// TwinCAT 3 PLC project Walking_Welding_Robot_Control_System
// ProgramVersion: 3.1.4020.4
// libraries:
//   Tc2_MC2, * (Beckhoff Automation GmbH)
//   Tc2_Standard, * (Beckhoff Automation GmbH)
//   Tc2_System, * (Beckhoff Automation GmbH)
//   Tc3_Module, * (Beckhoff Automation GmbH)
//   VisuDialogs, * (System)
// project tree:
//   DUTs/Axis/ Axis.TcPOU
//   DUTs/Filter_Current/ FB_Filter_Current_Hexapod_Robot.TcPOU, ST_Filter_Current_Hexapod_Robot_InitData.TcDUT, ST_Filter_Current_Hexapod_Robot_Input.TcDUT, ST_Filter_Current_Hexapod_Robot_Output.TcDUT
//   DUTs/Hexapod_Leg/ Hexapod_Leg.TcPOU (not stored)
//   DUTs/Mapping/ Leg_Control_Mapping_Model.TcPOU (not stored), Leg_Model_Mapping_Control.TcPOU (not stored), Variable_Control_Mapping_Model.TcPOU (not stored), Variable_Model_Mapping_Control.TcPOU (not stored)
//   DUTs/Robot_Simulink/ E_TcMatSimDataAreaType.TcDUT (not stored), FB_RobotWalking_OnEvenTerrain.TcPOU (not stored), FB_TcMatSimObject.TcPOU (not stored), ST_RobotWalking_OnEvenTerrain_InitData.TcDUT (not stored), ST_RobotWalking_OnEvenTerrain_Input.TcDUT (not stored), ST_RobotWalking_OnEvenTerrain_Output.TcDUT (not stored), ST_TcMatSimObjectDataAreaInfo.TcDUT (not stored)
//   DUTs/Touch_Signal_Detection/ FB_Tough_Signal_Detection_Simple.TcPOU, ST_Tough_Signal_Detection_Simple_InitData.TcDUT, ST_Tough_Signal_Detection_Simple_Input.TcDUT, ST_Tough_Signal_Detection_Simple_Output.TcDUT
//   DUTs/Welding_Arm_Simulink/ FB_WeldingArm6AxisMotion_Control.TcPOU, ST_WeldingArm6AxisMotion_Control_InitData.TcDUT, ST_WeldingArm6AxisMotion_Control_Input.TcDUT, ST_WeldingArm6AxisMotion_Control_Output.TcDUT
//   / GlobalTextList.TcGTLO, PlcTask.TcTTO, Sensor_Test.TcTTO, Simulink_Test.TcTTO, 视图管理器.TcVMO (not stored)
//   POUs/ Walking_Robot_Control.TcPOU, SignalData_Interface.TcPOU, Walking_Robot_Movement.TcPOU, Walking_Welding_Robot_Control.TcPOU, Welding_Arm_Control.TcPOU, Welding_Arm_Movement.TcPOU
//   VISUs/ ImagePool.TcIPO (not stored), Visu_Welding_Arm_Power.TcVIS, Visu_Welding_Arm_SimulinkMove.TcVIS, Visu_Walking_Robot_Home.TcVIS, Visu_Walking_Robot_Power.TcVIS, Visu_Walking_Robot_Reset.TcVIS, Visu_Walking_Robot_SimulinkMove.TcVIS, Visu_Walking_Robot_Stand.TcVIS, Visu_Walking_Welding_Robot_Control.TcVIS, Visu_Welcome.TcVIS, Visu_Welding_Arm_OldVersion.TcVIS
// real-time tasks:
//   TASK PlcTask: cycle T#4ms, priority 12, ADS port 350
//   TASK Simulink_Test: cycle T#4ms, priority 6, ADS port 351
//   TASK Sensor_Test: cycle T#1ms, priority 14, ADS port 352
//   TASK Walking_Welding_Robot_Task: cycle T#4ms, priority 10, ADS port 353
// motion (NC):
//   TASK NC-Task 1 SAF: cycle T#4ms, priority 4, ADS port 501
//   TASK NC-Task 1 SVB: cycle T#4ms, priority 8, ADS port 511
//   AXIS Axis 1 (id 1)
//     Velo: SlowManual=10, FastManual=20
//     OtherSettings: AllowMotionCmdToSlave=true, AllowMotionCmdToExtSetGenAxis=true
//     encoder EncType=19
//       EncPara: ScaleFactorNumerator=0.000152590218967, MaxCount=#xffffffff
//     drive DrvType=16
//       DrvPara: MaxCount=#xffffffff
//         TimeComp: TaskDelayCycles=1
//     controller CtrType=1
//       CtrPara: PriorControlFactor=1
//         Observer: BandWidth=20
//   AXIS Axis 2 (id 2)
//     Velo: SlowManual=10, FastManual=20
//     OtherSettings: AllowMotionCmdToSlave=true, AllowMotionCmdToExtSetGenAxis=true
//     encoder EncType=19
//       EncPara: ScaleFactorNumerator=0.000152590218967, MaxCount=#xffffffff
//     drive DrvType=16
//       DrvPara: MaxCount=#xffffffff
//         TimeComp: TaskDelayCycles=1
//     controller CtrType=1
//       CtrPara: PriorControlFactor=1
//         Observer: BandWidth=20
//   AXIS Axis 3 (id 3)
//     Velo: SlowManual=10, FastManual=20
//     OtherSettings: AllowMotionCmdToSlave=true, AllowMotionCmdToExtSetGenAxis=true
//     encoder EncType=19
//       EncPara: ScaleFactorNumerator=0.000152590218967, MaxCount=#xffffffff
//     drive DrvType=16
//       DrvPara: MaxCount=#xffffffff
//         TimeComp: TaskDelayCycles=1
//     controller CtrType=1
//       CtrPara: PriorControlFactor=1
//         Observer: BandWidth=20
//   AXIS Axis 4 (id 4)
//     Velo: SlowManual=10, FastManual=20
//     OtherSettings: AllowMotionCmdToSlave=true, AllowMotionCmdToExtSetGenAxis=true
//     encoder EncType=19
//       EncPara: ScaleFactorNumerator=0.000152590218967, MaxCount=#xffffffff
//     drive DrvType=16
//       DrvPara: MaxCount=#xffffffff
//         TimeComp: TaskDelayCycles=1
//     controller CtrType=1
//       CtrPara: PriorControlFactor=1
//         Observer: BandWidth=20
//   AXIS Axis 5 (id 5)
//     Velo: SlowManual=10, FastManual=20
//     OtherSettings: AllowMotionCmdToSlave=true, AllowMotionCmdToExtSetGenAxis=true
//     encoder EncType=19
//       EncPara: ScaleFactorNumerator=0.000152590218967, MaxCount=#xffffffff
//     drive DrvType=16
//       DrvPara: MaxCount=#xffffffff
//         TimeComp: TaskDelayCycles=1
//     controller CtrType=1
//       CtrPara: PriorControlFactor=1
//         Observer: BandWidth=20
//   AXIS Axis 6 (id 6)
//     Velo: SlowManual=10, FastManual=20
//     OtherSettings: AllowMotionCmdToSlave=true, AllowMotionCmdToExtSetGenAxis=true
//     encoder EncType=19
//       EncPara: ScaleFactorNumerator=0.000152590218967, MaxCount=#xffffffff
//     drive DrvType=16
//       DrvPara: MaxCount=#xffffffff
//         TimeComp: TaskDelayCycles=1
//     controller CtrType=1
//       CtrPara: PriorControlFactor=1
//         Observer: BandWidth=20
//   AXIS Axis 7 (id 7)
//     Velo: SlowManual=10, FastManual=20
//     OtherSettings: AllowMotionCmdToSlave=true, AllowMotionCmdToExtSetGenAxis=true
//     encoder EncType=19
//       EncPara: ScaleFactorNumerator=0.000152590218967, MaxCount=#xffffffff
//     drive DrvType=16
//       DrvPara: MaxCount=#xffffffff
//         TimeComp: TaskDelayCycles=1
//     controller CtrType=1
//       CtrPara: PriorControlFactor=1
//         Observer: BandWidth=20
//   AXIS Axis 8 (id 8)
//     Velo: SlowManual=10, FastManual=20
//     OtherSettings: AllowMotionCmdToSlave=true, AllowMotionCmdToExtSetGenAxis=true
//     encoder EncType=19
//       EncPara: ScaleFactorNumerator=0.000152590218967, MaxCount=#xffffffff
//     drive DrvType=16
//       DrvPara: MaxCount=#xffffffff
//         TimeComp: TaskDelayCycles=1
//     controller CtrType=1
//       CtrPara: PriorControlFactor=1
//         Observer: BandWidth=20
//   AXIS Axis 9 (id 9)
//     Velo: SlowManual=10, FastManual=20
//     OtherSettings: AllowMotionCmdToSlave=true, AllowMotionCmdToExtSetGenAxis=true
//     encoder EncType=19
//       EncPara: ScaleFactorNumerator=0.000152590218967, MaxCount=#xffffffff
//     drive DrvType=16
//       DrvPara: MaxCount=#xffffffff
//         TimeComp: TaskDelayCycles=1
//     controller CtrType=1
//       CtrPara: PriorControlFactor=1
//         Observer: BandWidth=20
//   AXIS Axis 10 (id 10)
//     Velo: SlowManual=10, FastManual=20
//     OtherSettings: AllowMotionCmdToSlave=true, AllowMotionCmdToExtSetGenAxis=true
//     encoder EncType=19
//       EncPara: ScaleFactorNumerator=0.000152590218967, MaxCount=#xffffffff
//     drive DrvType=16
//       DrvPara: MaxCount=#xffffffff
//         TimeComp: TaskDelayCycles=1
//     controller CtrType=1
//       CtrPara: PriorControlFactor=1
//         Observer: BandWidth=20
//   AXIS Axis 11 (id 11)
//     Velo: SlowManual=10, FastManual=20
//     OtherSettings: AllowMotionCmdToSlave=true, AllowMotionCmdToExtSetGenAxis=true
//     encoder EncType=19
//       EncPara: ScaleFactorNumerator=0.000152590218967, MaxCount=#xffffffff
//     drive DrvType=16
//       DrvPara: MaxCount=#xffffffff
//         TimeComp: TaskDelayCycles=1
//     controller CtrType=1
//       CtrPara: PriorControlFactor=1
//         Observer: BandWidth=20
//   AXIS Axis 12 (id 12)
//     Velo: SlowManual=10, FastManual=20
//     OtherSettings: AllowMotionCmdToSlave=true, AllowMotionCmdToExtSetGenAxis=true
//     encoder EncType=19
//       EncPara: ScaleFactorNumerator=0.000152590218967, MaxCount=#xffffffff
//     drive DrvType=16
//       DrvPara: MaxCount=#xffffffff
//         TimeComp: TaskDelayCycles=1
//     controller CtrType=1
//       CtrPara: PriorControlFactor=1
//         Observer: BandWidth=20
//   AXIS Axis 13 (id 13)
//     Velo: SlowManual=10, FastManual=20
//     OtherSettings: AllowMotionCmdToSlave=true, AllowMotionCmdToExtSetGenAxis=true
//     encoder EncType=19
//       EncPara: ScaleFactorNumerator=0.000152590218967, MaxCount=#xffffffff
//     drive DrvType=16
//       DrvPara: MaxCount=#xffffffff
//         TimeComp: TaskDelayCycles=1
//     controller CtrType=1
//       CtrPara: PriorControlFactor=1
//         Observer: BandWidth=20
//   AXIS Axis 14 (id 14)
//     Velo: SlowManual=10, FastManual=20
//     OtherSettings: AllowMotionCmdToSlave=true, AllowMotionCmdToExtSetGenAxis=true
//     encoder EncType=19
//       EncPara: ScaleFactorNumerator=0.000152590218967, MaxCount=#xffffffff
//     drive DrvType=16
//       DrvPara: MaxCount=#xffffffff
//         TimeComp: TaskDelayCycles=1
//     controller CtrType=1
//       CtrPara: PriorControlFactor=1
//         Observer: BandWidth=20
//   AXIS Axis 15 (id 15)
//     Velo: SlowManual=10, FastManual=20
//     OtherSettings: AllowMotionCmdToSlave=true, AllowMotionCmdToExtSetGenAxis=true
//     encoder EncType=19
//       EncPara: ScaleFactorNumerator=0.000152590218967, MaxCount=#xffffffff
//     drive DrvType=16
//       DrvPara: MaxCount=#xffffffff
//         TimeComp: TaskDelayCycles=1
//     controller CtrType=1
//       CtrPara: PriorControlFactor=1
//         Observer: BandWidth=20
//   AXIS Axis 16 (id 16)
//     Velo: SlowManual=10, FastManual=20
//     OtherSettings: AllowMotionCmdToSlave=true, AllowMotionCmdToExtSetGenAxis=true
//     encoder EncType=19
//       EncPara: ScaleFactorNumerator=0.000152590218967, MaxCount=#xffffffff
//     drive DrvType=16
//       DrvPara: MaxCount=#xffffffff
//         TimeComp: TaskDelayCycles=1
//     controller CtrType=1
//       CtrPara: PriorControlFactor=1
//         Observer: BandWidth=20
//   AXIS Axis 17 (id 17)
//     Velo: SlowManual=10, FastManual=20
//     OtherSettings: AllowMotionCmdToSlave=true, AllowMotionCmdToExtSetGenAxis=true
//     encoder EncType=19
//       EncPara: ScaleFactorNumerator=0.000152590218967, MaxCount=#xffffffff
//     drive DrvType=16
//       DrvPara: MaxCount=#xffffffff
//         TimeComp: TaskDelayCycles=1
//     controller CtrType=1
//       CtrPara: PriorControlFactor=1
//         Observer: BandWidth=20
//   AXIS Axis 18 (id 18)
//     Velo: SlowManual=10, FastManual=20
//     OtherSettings: AllowMotionCmdToSlave=true, AllowMotionCmdToExtSetGenAxis=true
//     encoder EncType=19
//       EncPara: ScaleFactorNumerator=0.000152590218967, MaxCount=#xffffffff
//     drive DrvType=16
//       DrvPara: MaxCount=#xffffffff
//         TimeComp: TaskDelayCycles=1
//     controller CtrType=1
//       CtrPara: PriorControlFactor=1
//         Observer: BandWidth=20
//   AXIS Axis 19 (id 19)
//     Velo: SlowManual=10, FastManual=20
//     OtherSettings: AllowMotionCmdToSlave=true
//     encoder EncType=19
//       EncPara: ScaleFactorNumerator=1.6954468774e-005, MaxCount=#xffffffff
//     drive DrvType=16
//       DrvPara: MaxCount=#xffffffff
//         TimeComp: TaskDelayCycles=1
//     controller CtrType=1
//       CtrPara: PriorControlFactor=1
//         Observer: BandWidth=20
//   AXIS Axis 20 (id 20)
//     Velo: SlowManual=10, FastManual=20
//     OtherSettings: AllowMotionCmdToSlave=true
//     encoder EncType=19
//       EncPara: ScaleFactorNumerator=0.006206896551724, MaxCount=#xffffffff
//     drive DrvType=16
//       DrvPara: MaxCount=#xffffffff
//         TimeComp: TaskDelayCycles=1
//     controller CtrType=1
//       CtrPara: PriorControlFactor=1
//         Observer: BandWidth=20
//   AXIS Axis 21 (id 21)
//     Velo: SlowManual=10, FastManual=20
//     OtherSettings: AllowMotionCmdToSlave=true
//     encoder EncType=19
//       EncPara: ScaleFactorNumerator=2.441443503e-006, MaxCount=#xffffffff
//     drive DrvType=16
//       DrvPara: MaxCount=#xffffffff
//         TimeComp: TaskDelayCycles=1
//     controller CtrType=1
//       CtrPara: PriorControlFactor=1
//         Observer: BandWidth=20
//   AXIS Axis 22 (id 22)
//     Velo: SlowManual=10, FastManual=20
//     OtherSettings: AllowMotionCmdToSlave=true
//     encoder EncType=19
//       EncPara: ScaleFactorNumerator=0.000365910901229, MaxCount=#xffffffff
//     drive DrvType=16
//       DrvPara: MaxCount=#xffffffff
//         TimeComp: TaskDelayCycles=1
//     controller CtrType=1
//       CtrPara: PriorControlFactor=1
//         Observer: BandWidth=20
//   AXIS Axis 23 (id 23)
//     Velo: SlowManual=10, FastManual=20
//     OtherSettings: AllowMotionCmdToSlave=true
//     encoder EncType=19
//       EncPara: ScaleFactorNumerator=0.000365910901229, MaxCount=#xffffffff
//     drive DrvType=16
//       DrvPara: MaxCount=#xffffffff
//         TimeComp: TaskDelayCycles=1
//     controller CtrType=1
//       CtrPara: PriorControlFactor=1
//         Observer: BandWidth=20
//   AXIS Axis 24 (id 24)
//     Velo: SlowManual=10, FastManual=20
//     OtherSettings: AllowMotionCmdToSlave=true
//     encoder EncType=19
//       EncPara: ScaleFactorNumerator=0.000365910901229, MaxCount=#xffffffff
//     drive DrvType=16
//       DrvPara: MaxCount=#xffffffff
//         TimeComp: TaskDelayCycles=1
//     controller CtrType=1
//       CtrPara: PriorControlFactor=1
//         Observer: BandWidth=20
// I/O:
//   DEVICE Device 3 (EtherCAT), AmsNetId 5.41.150.106.4.1
//     Drive 1 (Elmo Drive) [Gold EtherCAT GCON Drive Rev:0x000103F6]
//     Drive 2 (Elmo Drive) [Gold EtherCAT GCON Drive Rev:0x000103F6]
//     Drive 3 (Elmo Drive) [Gold EtherCAT GCON Drive Rev:0x000103F6]
//     Drive 4 (Elmo Drive) [Gold EtherCAT GCON Drive Rev:0x000103F6]
//     Drive 5 (Elmo Drive) [Gold EtherCAT GCON Drive Rev:0x000103F6]
//     Drive 6 (Elmo Drive) [Gold EtherCAT GCON Drive Rev:0x000103F6]
//     Drive 7 (Elmo Drive) [Gold EtherCAT GCON Drive Rev:0x000103F6]
//     Drive 8 (Elmo Drive) [Gold EtherCAT GCON Drive Rev:0x000103F6]
//     Drive 9 (Elmo Drive) [Gold EtherCAT GCON Drive Rev:0x000103F6]
//     Drive 10 (Elmo Drive) [Gold EtherCAT GCON Drive Rev:0x000103F6]
//     Drive 11 (Elmo Drive) [Gold EtherCAT GCON Drive Rev:0x000103F6]
//     Drive 12 (Elmo Drive) [Gold EtherCAT GCON Drive Rev:0x000103F6]
//     Drive 13 (Elmo Drive) [Gold EtherCAT GCON Drive Rev:0x000103F6]
//     Drive 14 (Elmo Drive) [Gold EtherCAT GCON Drive Rev:0x000103F6]
//     Drive 15 (Elmo Drive) [Gold EtherCAT GCON Drive Rev:0x000103F6]
//     Drive 16 (Elmo Drive) [Gold EtherCAT GCON Drive Rev:0x000103F6]
//     Drive 17 (Elmo Drive) [Gold EtherCAT GCON Drive Rev:0x000103F6]
//     Drive 18 (Elmo Drive) [Gold EtherCAT GCON Drive Rev:0x000103F6]
//     Drive 37 (Elmo Drive) [Gold EtherCAT GCON Drive Rev:0x000103F6]
//     Drive 38 (Elmo Drive) [Gold EtherCAT GCON Drive Rev:0x000103F6]
//     Drive 39 (Elmo Drive) [Gold EtherCAT GCON Drive Rev:0x000103F6]
//     Drive 40 (Elmo Drive) [Gold EtherCAT GCON Drive Rev:0x000103F6]
//     Drive 41 (Elmo Drive) [Gold EtherCAT GCON Drive Rev:0x000103F6]
//     Drive 42 (Elmo Drive) [Gold EtherCAT GCON Drive Rev:0x000103F6]
// variable links:
//   NC-Task 1 SAF/Axes/Axis 1 <-> Device 3 (EtherCAT)/Drive 1 (Elmo Drive)
//     Drive/Inputs/In/nDcOutputTime <-> InfoData/DcOutputShift
//     Drive/Inputs/In/nState1 <-> Inputs/Status word
//     Drive/Inputs/In/nState2 <-> Inputs/Status word @bit 8
//     Drive/Inputs/In/nState4 @bit 1 <-> WcState/InputToggle
//     Drive/Inputs/In/nState4 <-> WcState/WcState
//     Drive/Outputs/Out/nCtrl1 <-> Outputs/Control word
//     Drive/Outputs/Out/nCtrl2 <-> Outputs/Control word @bit 8
//     Drive/Outputs/Out/nDataOut1 <-> Outputs/Target Position
//     Enc/Inputs/In/nDataIn1 <-> Inputs/Position actual value
//     Enc/Inputs/In/nDcInputTime <-> InfoData/DcInputShift
//     Enc/Inputs/In/nState4 @bit 1 <-> WcState/InputToggle
//     Enc/Inputs/In/nState4 <-> WcState/WcState
//   NC-Task 1 SAF/Axes/Axis 10 <-> Device 3 (EtherCAT)/Drive 10 (Elmo Drive)
//     Drive/Inputs/In/nDcOutputTime <-> InfoData/DcOutputShift
//     Drive/Inputs/In/nState1 <-> Inputs/Status word
//     Drive/Inputs/In/nState2 <-> Inputs/Status word @bit 8
//     Drive/Inputs/In/nState4 @bit 1 <-> WcState/InputToggle
//     Drive/Inputs/In/nState4 <-> WcState/WcState
//     Drive/Outputs/Out/nCtrl1 <-> Outputs/Control word
//     Drive/Outputs/Out/nCtrl2 <-> Outputs/Control word @bit 8
//     Drive/Outputs/Out/nDataOut1 <-> Outputs/Target Position
//     Enc/Inputs/In/nDataIn1 <-> Inputs/Position actual value
//     Enc/Inputs/In/nDcInputTime <-> InfoData/DcInputShift
//     Enc/Inputs/In/nState4 @bit 1 <-> WcState/InputToggle
//     Enc/Inputs/In/nState4 <-> WcState/WcState
//   NC-Task 1 SAF/Axes/Axis 11 <-> Device 3 (EtherCAT)/Drive 11 (Elmo Drive)
//     Drive/Inputs/In/nDcOutputTime <-> InfoData/DcOutputShift
//     Drive/Inputs/In/nState1 <-> Inputs/Status word
//     Drive/Inputs/In/nState2 <-> Inputs/Status word @bit 8
//     Drive/Inputs/In/nState4 @bit 1 <-> WcState/InputToggle
//     Drive/Inputs/In/nState4 <-> WcState/WcState
//     Drive/Outputs/Out/nCtrl1 <-> Outputs/Control word
//     Drive/Outputs/Out/nCtrl2 <-> Outputs/Control word @bit 8
//     Drive/Outputs/Out/nDataOut1 <-> Outputs/Target Position
//     Enc/Inputs/In/nDataIn1 <-> Inputs/Position actual value
//     Enc/Inputs/In/nDcInputTime <-> InfoData/DcInputShift
//     Enc/Inputs/In/nState4 @bit 1 <-> WcState/InputToggle
//     Enc/Inputs/In/nState4 <-> WcState/WcState
//   NC-Task 1 SAF/Axes/Axis 12 <-> Device 3 (EtherCAT)/Drive 12 (Elmo Drive)
//     Drive/Inputs/In/nDcOutputTime <-> InfoData/DcOutputShift
//     Drive/Inputs/In/nState1 <-> Inputs/Status word
//     Drive/Inputs/In/nState2 <-> Inputs/Status word @bit 8
//     Drive/Inputs/In/nState4 @bit 1 <-> WcState/InputToggle
//     Drive/Inputs/In/nState4 <-> WcState/WcState
//     Drive/Outputs/Out/nCtrl1 <-> Outputs/Control word
//     Drive/Outputs/Out/nCtrl2 <-> Outputs/Control word @bit 8
//     Drive/Outputs/Out/nDataOut1 <-> Outputs/Target Position
//     Enc/Inputs/In/nDataIn1 <-> Inputs/Position actual value
//     Enc/Inputs/In/nDcInputTime <-> InfoData/DcInputShift
//     Enc/Inputs/In/nState4 @bit 1 <-> WcState/InputToggle
//     Enc/Inputs/In/nState4 <-> WcState/WcState
//   NC-Task 1 SAF/Axes/Axis 13 <-> Device 3 (EtherCAT)/Drive 13 (Elmo Drive)
//     Drive/Inputs/In/nDcOutputTime <-> InfoData/DcOutputShift
//     Drive/Inputs/In/nState1 <-> Inputs/Status word
//     Drive/Inputs/In/nState2 <-> Inputs/Status word @bit 8
//     Drive/Inputs/In/nState4 @bit 1 <-> WcState/InputToggle
//     Drive/Inputs/In/nState4 <-> WcState/WcState
//     Drive/Outputs/Out/nCtrl1 <-> Outputs/Control word
//     Drive/Outputs/Out/nCtrl2 <-> Outputs/Control word @bit 8
//     Drive/Outputs/Out/nDataOut1 <-> Outputs/Target Position
//     Enc/Inputs/In/nDataIn1 <-> Inputs/Position actual value
//     Enc/Inputs/In/nDcInputTime <-> InfoData/DcInputShift
//     Enc/Inputs/In/nState4 @bit 1 <-> WcState/InputToggle
//     Enc/Inputs/In/nState4 <-> WcState/WcState
//   NC-Task 1 SAF/Axes/Axis 14 <-> Device 3 (EtherCAT)/Drive 14 (Elmo Drive)
//     Drive/Inputs/In/nDcOutputTime <-> InfoData/DcOutputShift
//     Drive/Inputs/In/nState1 <-> Inputs/Status word
//     Drive/Inputs/In/nState2 <-> Inputs/Status word @bit 8
//     Drive/Inputs/In/nState4 @bit 1 <-> WcState/InputToggle
//     Drive/Inputs/In/nState4 <-> WcState/WcState
//     Drive/Outputs/Out/nCtrl1 <-> Outputs/Control word
//     Drive/Outputs/Out/nCtrl2 <-> Outputs/Control word @bit 8
//     Drive/Outputs/Out/nDataOut1 <-> Outputs/Target Position
//     Enc/Inputs/In/nDataIn1 <-> Inputs/Position actual value
//     Enc/Inputs/In/nDcInputTime <-> InfoData/DcInputShift
//     Enc/Inputs/In/nState4 @bit 1 <-> WcState/InputToggle
//     Enc/Inputs/In/nState4 <-> WcState/WcState
//   NC-Task 1 SAF/Axes/Axis 15 <-> Device 3 (EtherCAT)/Drive 15 (Elmo Drive)
//     Drive/Inputs/In/nDcOutputTime <-> InfoData/DcOutputShift
//     Drive/Inputs/In/nState1 <-> Inputs/Status word
//     Drive/Inputs/In/nState2 <-> Inputs/Status word @bit 8
//     Drive/Inputs/In/nState4 @bit 1 <-> WcState/InputToggle
//     Drive/Inputs/In/nState4 <-> WcState/WcState
//     Drive/Outputs/Out/nCtrl1 <-> Outputs/Control word
//     Drive/Outputs/Out/nCtrl2 <-> Outputs/Control word @bit 8
//     Drive/Outputs/Out/nDataOut1 <-> Outputs/Target Position
//     Enc/Inputs/In/nDataIn1 <-> Inputs/Position actual value
//     Enc/Inputs/In/nDcInputTime <-> InfoData/DcInputShift
//     Enc/Inputs/In/nState4 @bit 1 <-> WcState/InputToggle
//     Enc/Inputs/In/nState4 <-> WcState/WcState
//   NC-Task 1 SAF/Axes/Axis 16 <-> Device 3 (EtherCAT)/Drive 16 (Elmo Drive)
//     Drive/Inputs/In/nDcOutputTime <-> InfoData/DcOutputShift
//     Drive/Inputs/In/nState1 <-> Inputs/Status word
//     Drive/Inputs/In/nState2 <-> Inputs/Status word @bit 8
//     Drive/Inputs/In/nState4 @bit 1 <-> WcState/InputToggle
//     Drive/Inputs/In/nState4 <-> WcState/WcState
//     Drive/Outputs/Out/nCtrl1 <-> Outputs/Control word
//     Drive/Outputs/Out/nCtrl2 <-> Outputs/Control word @bit 8
//     Drive/Outputs/Out/nDataOut1 <-> Outputs/Target Position
//     Enc/Inputs/In/nDataIn1 <-> Inputs/Position actual value
//     Enc/Inputs/In/nDcInputTime <-> InfoData/DcInputShift
//     Enc/Inputs/In/nState4 @bit 1 <-> WcState/InputToggle
//     Enc/Inputs/In/nState4 <-> WcState/WcState
//   NC-Task 1 SAF/Axes/Axis 17 <-> Device 3 (EtherCAT)/Drive 17 (Elmo Drive)
//     Drive/Inputs/In/nDcOutputTime <-> InfoData/DcOutputShift
//     Drive/Inputs/In/nState1 <-> Inputs/Status word
//     Drive/Inputs/In/nState2 <-> Inputs/Status word @bit 8
//     Drive/Inputs/In/nState4 @bit 1 <-> WcState/InputToggle
//     Drive/Inputs/In/nState4 <-> WcState/WcState
//     Drive/Outputs/Out/nCtrl1 <-> Outputs/Control word
//     Drive/Outputs/Out/nCtrl2 <-> Outputs/Control word @bit 8
//     Drive/Outputs/Out/nDataOut1 <-> Outputs/Target Position
//     Enc/Inputs/In/nDataIn1 <-> Inputs/Position actual value
//     Enc/Inputs/In/nDcInputTime <-> InfoData/DcInputShift
//     Enc/Inputs/In/nState4 @bit 1 <-> WcState/InputToggle
//     Enc/Inputs/In/nState4 <-> WcState/WcState
//   NC-Task 1 SAF/Axes/Axis 18 <-> Device 3 (EtherCAT)/Drive 18 (Elmo Drive)
//     Drive/Inputs/In/nDcOutputTime <-> InfoData/DcOutputShift
//     Drive/Inputs/In/nState1 <-> Inputs/Status word
//     Drive/Inputs/In/nState2 <-> Inputs/Status word @bit 8
//     Drive/Inputs/In/nState4 @bit 1 <-> WcState/InputToggle
//     Drive/Inputs/In/nState4 <-> WcState/WcState
//     Drive/Outputs/Out/nCtrl1 <-> Outputs/Control word
//     Drive/Outputs/Out/nCtrl2 <-> Outputs/Control word @bit 8
//     Drive/Outputs/Out/nDataOut1 <-> Outputs/Target Position
//     Enc/Inputs/In/nDataIn1 <-> Inputs/Position actual value
//     Enc/Inputs/In/nDcInputTime <-> InfoData/DcInputShift
//     Enc/Inputs/In/nState4 @bit 1 <-> WcState/InputToggle
//     Enc/Inputs/In/nState4 <-> WcState/WcState
//   NC-Task 1 SAF/Axes/Axis 19 <-> Device 3 (EtherCAT)/Drive 37 (Elmo Drive)
//     Drive/Inputs/In/nDcOutputTime <-> InfoData/DcOutputShift
//     Drive/Inputs/In/nState1 <-> Inputs/Status word
//     Drive/Inputs/In/nState2 <-> Inputs/Status word @bit 8
//     Drive/Inputs/In/nState4 @bit 1 <-> WcState/InputToggle
//     Drive/Inputs/In/nState4 <-> WcState/WcState
//     Drive/Outputs/Out/nCtrl1 <-> Outputs/Control word
//     Drive/Outputs/Out/nCtrl2 <-> Outputs/Control word @bit 8
//     Drive/Outputs/Out/nDataOut1 <-> Outputs/Target Position
//     Enc/Inputs/In/nDataIn1 <-> Inputs/Position actual value
//     Enc/Inputs/In/nDcInputTime <-> InfoData/DcInputShift
//     Enc/Inputs/In/nState4 @bit 1 <-> WcState/InputToggle
//     Enc/Inputs/In/nState4 <-> WcState/WcState
//   NC-Task 1 SAF/Axes/Axis 2 <-> Device 3 (EtherCAT)/Drive 2 (Elmo Drive)
//     Drive/Inputs/In/nDcOutputTime <-> InfoData/DcOutputShift
//     Drive/Inputs/In/nState1 <-> Inputs/Status word
//     Drive/Inputs/In/nState2 <-> Inputs/Status word @bit 8
//     Drive/Inputs/In/nState4 @bit 1 <-> WcState/InputToggle
//     Drive/Inputs/In/nState4 <-> WcState/WcState
//     Drive/Outputs/Out/nCtrl1 <-> Outputs/Control word
//     Drive/Outputs/Out/nCtrl2 <-> Outputs/Control word @bit 8
//     Drive/Outputs/Out/nDataOut1 <-> Outputs/Target Position
//     Enc/Inputs/In/nDataIn1 <-> Inputs/Position actual value
//     Enc/Inputs/In/nDcInputTime <-> InfoData/DcInputShift
//     Enc/Inputs/In/nState4 @bit 1 <-> WcState/InputToggle
//     Enc/Inputs/In/nState4 <-> WcState/WcState
//   NC-Task 1 SAF/Axes/Axis 20 <-> Device 3 (EtherCAT)/Drive 38 (Elmo Drive)
//     Drive/Inputs/In/nDcOutputTime <-> InfoData/DcOutputShift
//     Drive/Inputs/In/nState1 <-> Inputs/Status word
//     Drive/Inputs/In/nState2 <-> Inputs/Status word @bit 8
//     Drive/Inputs/In/nState4 @bit 1 <-> WcState/InputToggle
//     Drive/Inputs/In/nState4 <-> WcState/WcState
//     Drive/Outputs/Out/nCtrl1 <-> Outputs/Control word
//     Drive/Outputs/Out/nCtrl2 <-> Outputs/Control word @bit 8
//     Drive/Outputs/Out/nDataOut1 <-> Outputs/Target Position
//     Enc/Inputs/In/nDataIn1 <-> Inputs/Position actual value
//     Enc/Inputs/In/nDcInputTime <-> InfoData/DcInputShift
//     Enc/Inputs/In/nState4 @bit 1 <-> WcState/InputToggle
//     Enc/Inputs/In/nState4 <-> WcState/WcState
//   NC-Task 1 SAF/Axes/Axis 21 <-> Device 3 (EtherCAT)/Drive 39 (Elmo Drive)
//     Drive/Inputs/In/nDcOutputTime <-> InfoData/DcOutputShift
//     Drive/Inputs/In/nState1 <-> Inputs/Status word
//     Drive/Inputs/In/nState2 <-> Inputs/Status word @bit 8
//     Drive/Inputs/In/nState4 @bit 1 <-> WcState/InputToggle
//     Drive/Inputs/In/nState4 <-> WcState/WcState
//     Drive/Outputs/Out/nCtrl1 <-> Outputs/Control word
//     Drive/Outputs/Out/nCtrl2 <-> Outputs/Control word @bit 8
//     Drive/Outputs/Out/nDataOut1 <-> Outputs/Target Position
//     Enc/Inputs/In/nDataIn1 <-> Inputs/Position actual value
//     Enc/Inputs/In/nDcInputTime <-> InfoData/DcInputShift
//     Enc/Inputs/In/nState4 @bit 1 <-> WcState/InputToggle
//     Enc/Inputs/In/nState4 <-> WcState/WcState
//   NC-Task 1 SAF/Axes/Axis 22 <-> Device 3 (EtherCAT)/Drive 40 (Elmo Drive)
//     Drive/Inputs/In/nDcOutputTime <-> InfoData/DcOutputShift
//     Drive/Inputs/In/nState1 <-> Inputs/Status word
//     Drive/Inputs/In/nState2 <-> Inputs/Status word @bit 8
//     Drive/Inputs/In/nState4 @bit 1 <-> WcState/InputToggle
//     Drive/Inputs/In/nState4 <-> WcState/WcState
//     Drive/Outputs/Out/nCtrl1 <-> Outputs/Control word
//     Drive/Outputs/Out/nCtrl2 <-> Outputs/Control word @bit 8
//     Drive/Outputs/Out/nDataOut1 <-> Outputs/Target Position
//     Enc/Inputs/In/nDataIn1 <-> Inputs/Position actual value
//     Enc/Inputs/In/nDcInputTime <-> InfoData/DcInputShift
//     Enc/Inputs/In/nState4 @bit 1 <-> WcState/InputToggle
//     Enc/Inputs/In/nState4 <-> WcState/WcState
//   NC-Task 1 SAF/Axes/Axis 23 <-> Device 3 (EtherCAT)/Drive 41 (Elmo Drive)
//     Drive/Inputs/In/nDcOutputTime <-> InfoData/DcOutputShift
//     Drive/Inputs/In/nState1 <-> Inputs/Status word
//     Drive/Inputs/In/nState2 <-> Inputs/Status word @bit 8
//     Drive/Inputs/In/nState4 @bit 1 <-> WcState/InputToggle
//     Drive/Inputs/In/nState4 <-> WcState/WcState
//     Drive/Outputs/Out/nCtrl1 <-> Outputs/Control word
//     Drive/Outputs/Out/nCtrl2 <-> Outputs/Control word @bit 8
//     Drive/Outputs/Out/nDataOut1 <-> Outputs/Target Position
//     Enc/Inputs/In/nDataIn1 <-> Inputs/Position actual value
//     Enc/Inputs/In/nDcInputTime <-> InfoData/DcInputShift
//     Enc/Inputs/In/nState4 @bit 1 <-> WcState/InputToggle
//     Enc/Inputs/In/nState4 <-> WcState/WcState
//   NC-Task 1 SAF/Axes/Axis 24 <-> Device 3 (EtherCAT)/Drive 42 (Elmo Drive)
//     Drive/Inputs/In/nDcOutputTime <-> InfoData/DcOutputShift
//     Drive/Inputs/In/nState1 <-> Inputs/Status word
//     Drive/Inputs/In/nState2 <-> Inputs/Status word @bit 8
//     Drive/Inputs/In/nState4 @bit 1 <-> WcState/InputToggle
//     Drive/Inputs/In/nState4 <-> WcState/WcState
//     Drive/Outputs/Out/nCtrl1 <-> Outputs/Control word
//     Drive/Outputs/Out/nCtrl2 <-> Outputs/Control word @bit 8
//     Drive/Outputs/Out/nDataOut1 <-> Outputs/Target Position
//     Enc/Inputs/In/nDataIn1 <-> Inputs/Position actual value
//     Enc/Inputs/In/nDcInputTime <-> InfoData/DcInputShift
//     Enc/Inputs/In/nState4 @bit 1 <-> WcState/InputToggle
//     Enc/Inputs/In/nState4 <-> WcState/WcState
//   NC-Task 1 SAF/Axes/Axis 3 <-> Device 3 (EtherCAT)/Drive 3 (Elmo Drive)
//     Drive/Inputs/In/nDcOutputTime <-> InfoData/DcOutputShift
//     Drive/Inputs/In/nState1 <-> Inputs/Status word
//     Drive/Inputs/In/nState2 <-> Inputs/Status word @bit 8
//     Drive/Inputs/In/nState4 @bit 1 <-> WcState/InputToggle
//     Drive/Inputs/In/nState4 <-> WcState/WcState
//     Drive/Outputs/Out/nCtrl1 <-> Outputs/Control word
//     Drive/Outputs/Out/nCtrl2 <-> Outputs/Control word @bit 8
//     Drive/Outputs/Out/nDataOut1 <-> Outputs/Target Position
//     Enc/Inputs/In/nDataIn1 <-> Inputs/Position actual value
//     Enc/Inputs/In/nDcInputTime <-> InfoData/DcInputShift
//     Enc/Inputs/In/nState4 @bit 1 <-> WcState/InputToggle
//     Enc/Inputs/In/nState4 <-> WcState/WcState
//   NC-Task 1 SAF/Axes/Axis 4 <-> Device 3 (EtherCAT)/Drive 4 (Elmo Drive)
//     Drive/Inputs/In/nDcOutputTime <-> InfoData/DcOutputShift
//     Drive/Inputs/In/nState1 <-> Inputs/Status word
//     Drive/Inputs/In/nState2 <-> Inputs/Status word @bit 8
//     Drive/Inputs/In/nState4 @bit 1 <-> WcState/InputToggle
//     Drive/Inputs/In/nState4 <-> WcState/WcState
//     Drive/Outputs/Out/nCtrl1 <-> Outputs/Control word
//     Drive/Outputs/Out/nCtrl2 <-> Outputs/Control word @bit 8
//     Drive/Outputs/Out/nDataOut1 <-> Outputs/Target Position
//     Enc/Inputs/In/nDataIn1 <-> Inputs/Position actual value
//     Enc/Inputs/In/nDcInputTime <-> InfoData/DcInputShift
//     Enc/Inputs/In/nState4 @bit 1 <-> WcState/InputToggle
//     Enc/Inputs/In/nState4 <-> WcState/WcState
//   NC-Task 1 SAF/Axes/Axis 5 <-> Device 3 (EtherCAT)/Drive 5 (Elmo Drive)
//     Drive/Inputs/In/nDcOutputTime <-> InfoData/DcOutputShift
//     Drive/Inputs/In/nState1 <-> Inputs/Status word
//     Drive/Inputs/In/nState2 <-> Inputs/Status word @bit 8
//     Drive/Inputs/In/nState4 @bit 1 <-> WcState/InputToggle
//     Drive/Inputs/In/nState4 <-> WcState/WcState
//     Drive/Outputs/Out/nCtrl1 <-> Outputs/Control word
//     Drive/Outputs/Out/nCtrl2 <-> Outputs/Control word @bit 8
//     Drive/Outputs/Out/nDataOut1 <-> Outputs/Target Position
//     Enc/Inputs/In/nDataIn1 <-> Inputs/Position actual value
//     Enc/Inputs/In/nDcInputTime <-> InfoData/DcInputShift
//     Enc/Inputs/In/nState4 @bit 1 <-> WcState/InputToggle
//     Enc/Inputs/In/nState4 <-> WcState/WcState
//   NC-Task 1 SAF/Axes/Axis 6 <-> Device 3 (EtherCAT)/Drive 6 (Elmo Drive)
//     Drive/Inputs/In/nDcOutputTime <-> InfoData/DcOutputShift
//     Drive/Inputs/In/nState1 <-> Inputs/Status word
//     Drive/Inputs/In/nState2 <-> Inputs/Status word @bit 8
//     Drive/Inputs/In/nState4 @bit 1 <-> WcState/InputToggle
//     Drive/Inputs/In/nState4 <-> WcState/WcState
//     Drive/Outputs/Out/nCtrl1 <-> Outputs/Control word
//     Drive/Outputs/Out/nCtrl2 <-> Outputs/Control word @bit 8
//     Drive/Outputs/Out/nDataOut1 <-> Outputs/Target Position
//     Enc/Inputs/In/nDataIn1 <-> Inputs/Position actual value
//     Enc/Inputs/In/nDcInputTime <-> InfoData/DcInputShift
//     Enc/Inputs/In/nState4 @bit 1 <-> WcState/InputToggle
//     Enc/Inputs/In/nState4 <-> WcState/WcState
//   NC-Task 1 SAF/Axes/Axis 7 <-> Device 3 (EtherCAT)/Drive 7 (Elmo Drive)
//     Drive/Inputs/In/nDcOutputTime <-> InfoData/DcOutputShift
//     Drive/Inputs/In/nState1 <-> Inputs/Status word
//     Drive/Inputs/In/nState2 <-> Inputs/Status word @bit 8
//     Drive/Inputs/In/nState4 @bit 1 <-> WcState/InputToggle
//     Drive/Inputs/In/nState4 <-> WcState/WcState
//     Drive/Outputs/Out/nCtrl1 <-> Outputs/Control word
//     Drive/Outputs/Out/nCtrl2 <-> Outputs/Control word @bit 8
//     Drive/Outputs/Out/nDataOut1 <-> Outputs/Target Position
//     Enc/Inputs/In/nDataIn1 <-> Inputs/Position actual value
//     Enc/Inputs/In/nDcInputTime <-> InfoData/DcInputShift
//     Enc/Inputs/In/nState4 @bit 1 <-> WcState/InputToggle
//     Enc/Inputs/In/nState4 <-> WcState/WcState
//   NC-Task 1 SAF/Axes/Axis 8 <-> Device 3 (EtherCAT)/Drive 8 (Elmo Drive)
//     Drive/Inputs/In/nDcOutputTime <-> InfoData/DcOutputShift
//     Drive/Inputs/In/nState1 <-> Inputs/Status word
//     Drive/Inputs/In/nState2 <-> Inputs/Status word @bit 8
//     Drive/Inputs/In/nState4 @bit 1 <-> WcState/InputToggle
//     Drive/Inputs/In/nState4 <-> WcState/WcState
//     Drive/Outputs/Out/nCtrl1 <-> Outputs/Control word
//     Drive/Outputs/Out/nCtrl2 <-> Outputs/Control word @bit 8
//     Drive/Outputs/Out/nDataOut1 <-> Outputs/Target Position
//     Enc/Inputs/In/nDataIn1 <-> Inputs/Position actual value
//     Enc/Inputs/In/nDcInputTime <-> InfoData/DcInputShift
//     Enc/Inputs/In/nState4 @bit 1 <-> WcState/InputToggle
//     Enc/Inputs/In/nState4 <-> WcState/WcState
//   NC-Task 1 SAF/Axes/Axis 9 <-> Device 3 (EtherCAT)/Drive 9 (Elmo Drive)
//     Drive/Inputs/In/nDcOutputTime <-> InfoData/DcOutputShift
//     Drive/Inputs/In/nState1 <-> Inputs/Status word
//     Drive/Inputs/In/nState2 <-> Inputs/Status word @bit 8
//     Drive/Inputs/In/nState4 @bit 1 <-> WcState/InputToggle
//     Drive/Inputs/In/nState4 <-> WcState/WcState
//     Drive/Outputs/Out/nCtrl1 <-> Outputs/Control word
//     Drive/Outputs/Out/nCtrl2 <-> Outputs/Control word @bit 8
//     Drive/Outputs/Out/nDataOut1 <-> Outputs/Target Position
//     Enc/Inputs/In/nDataIn1 <-> Inputs/Position actual value
//     Enc/Inputs/In/nDcInputTime <-> InfoData/DcInputShift
//     Enc/Inputs/In/nState4 @bit 1 <-> WcState/InputToggle
//     Enc/Inputs/In/nState4 <-> WcState/WcState
//   Walking_Welding_Robot_Control_System/Walking_Welding_Robot_Control_System Instance <-> Device 3 (EtherCAT)/Drive 1 (Elmo Drive)
//     Simulink_Test Inputs/Walking_Robot_Control.Current_Turque_Value[1] <-> Inputs_1/Current actual value
//   Walking_Welding_Robot_Control_System/Walking_Welding_Robot_Control_System Instance <-> Device 3 (EtherCAT)/Drive 10 (Elmo Drive)
//     Simulink_Test Inputs/Walking_Robot_Control.Current_Turque_Value[10] <-> Inputs_1/Current actual value
//   Walking_Welding_Robot_Control_System/Walking_Welding_Robot_Control_System Instance <-> Device 3 (EtherCAT)/Drive 11 (Elmo Drive)
//     Simulink_Test Inputs/Walking_Robot_Control.Current_Turque_Value[11] <-> Inputs_1/Current actual value
//   Walking_Welding_Robot_Control_System/Walking_Welding_Robot_Control_System Instance <-> Device 3 (EtherCAT)/Drive 12 (Elmo Drive)
//     Simulink_Test Inputs/Walking_Robot_Control.Current_Turque_Value[12] <-> Inputs_1/Current actual value
//   Walking_Welding_Robot_Control_System/Walking_Welding_Robot_Control_System Instance <-> Device 3 (EtherCAT)/Drive 13 (Elmo Drive)
//     Simulink_Test Inputs/Walking_Robot_Control.Current_Turque_Value[13] <-> Inputs_1/Current actual value
//   Walking_Welding_Robot_Control_System/Walking_Welding_Robot_Control_System Instance <-> Device 3 (EtherCAT)/Drive 14 (Elmo Drive)
//     Simulink_Test Inputs/Walking_Robot_Control.Current_Turque_Value[14] <-> Inputs_1/Current actual value
//   Walking_Welding_Robot_Control_System/Walking_Welding_Robot_Control_System Instance <-> Device 3 (EtherCAT)/Drive 15 (Elmo Drive)
//     Simulink_Test Inputs/Walking_Robot_Control.Current_Turque_Value[15] <-> Inputs_1/Current actual value
//   Walking_Welding_Robot_Control_System/Walking_Welding_Robot_Control_System Instance <-> Device 3 (EtherCAT)/Drive 16 (Elmo Drive)
//     Simulink_Test Inputs/Walking_Robot_Control.Current_Turque_Value[16] <-> Inputs_1/Current actual value
//   Walking_Welding_Robot_Control_System/Walking_Welding_Robot_Control_System Instance <-> Device 3 (EtherCAT)/Drive 17 (Elmo Drive)
//     Simulink_Test Inputs/Walking_Robot_Control.Current_Turque_Value[17] <-> Inputs_1/Current actual value
//   Walking_Welding_Robot_Control_System/Walking_Welding_Robot_Control_System Instance <-> Device 3 (EtherCAT)/Drive 18 (Elmo Drive)
//     Simulink_Test Inputs/Walking_Robot_Control.Current_Turque_Value[18] <-> Inputs_1/Current actual value
//   Walking_Welding_Robot_Control_System/Walking_Welding_Robot_Control_System Instance <-> Device 3 (EtherCAT)/Drive 2 (Elmo Drive)
//     Simulink_Test Inputs/Walking_Robot_Control.Current_Turque_Value[2] <-> Inputs_1/Current actual value
//   Walking_Welding_Robot_Control_System/Walking_Welding_Robot_Control_System Instance <-> Device 3 (EtherCAT)/Drive 3 (Elmo Drive)
//     Simulink_Test Inputs/Walking_Robot_Control.Current_Turque_Value[3] <-> Inputs_1/Current actual value
//   Walking_Welding_Robot_Control_System/Walking_Welding_Robot_Control_System Instance <-> Device 3 (EtherCAT)/Drive 37 (Elmo Drive)
//     PlcTask Inputs/Welding_Arm_Control.Digital_Inputs[1] <-> Inputs/Digital Inputs
//   Walking_Welding_Robot_Control_System/Walking_Welding_Robot_Control_System Instance <-> Device 3 (EtherCAT)/Drive 38 (Elmo Drive)
//     PlcTask Inputs/Welding_Arm_Control.Digital_Inputs[2] <-> Inputs/Digital Inputs
//   Walking_Welding_Robot_Control_System/Walking_Welding_Robot_Control_System Instance <-> Device 3 (EtherCAT)/Drive 39 (Elmo Drive)
//     PlcTask Inputs/Welding_Arm_Control.Digital_Inputs[3] <-> Inputs/Digital Inputs
//   Walking_Welding_Robot_Control_System/Walking_Welding_Robot_Control_System Instance <-> Device 3 (EtherCAT)/Drive 4 (Elmo Drive)
//     Simulink_Test Inputs/Walking_Robot_Control.Current_Turque_Value[4] <-> Inputs_1/Current actual value
//   Walking_Welding_Robot_Control_System/Walking_Welding_Robot_Control_System Instance <-> Device 3 (EtherCAT)/Drive 40 (Elmo Drive)
//     PlcTask Inputs/Welding_Arm_Control.Digital_Inputs[4] <-> Inputs/Digital Inputs
//   Walking_Welding_Robot_Control_System/Walking_Welding_Robot_Control_System Instance <-> Device 3 (EtherCAT)/Drive 41 (Elmo Drive)
//     PlcTask Inputs/Welding_Arm_Control.Digital_Inputs[5] <-> Inputs/Digital Inputs
//   Walking_Welding_Robot_Control_System/Walking_Welding_Robot_Control_System Instance <-> Device 3 (EtherCAT)/Drive 42 (Elmo Drive)
//     PlcTask Inputs/Welding_Arm_Control.Digital_Inputs[6] <-> Inputs/Digital Inputs
//   Walking_Welding_Robot_Control_System/Walking_Welding_Robot_Control_System Instance <-> Device 3 (EtherCAT)/Drive 5 (Elmo Drive)
//     Simulink_Test Inputs/Walking_Robot_Control.Current_Turque_Value[5] <-> Inputs_1/Current actual value
//   Walking_Welding_Robot_Control_System/Walking_Welding_Robot_Control_System Instance <-> Device 3 (EtherCAT)/Drive 6 (Elmo Drive)
//     Simulink_Test Inputs/Walking_Robot_Control.Current_Turque_Value[6] <-> Inputs_1/Current actual value
//   Walking_Welding_Robot_Control_System/Walking_Welding_Robot_Control_System Instance <-> Device 3 (EtherCAT)/Drive 7 (Elmo Drive)
//     Simulink_Test Inputs/Walking_Robot_Control.Current_Turque_Value[7] <-> Inputs_1/Current actual value
//   Walking_Welding_Robot_Control_System/Walking_Welding_Robot_Control_System Instance <-> Device 3 (EtherCAT)/Drive 8 (Elmo Drive)
//     Simulink_Test Inputs/Walking_Robot_Control.Current_Turque_Value[8] <-> Inputs_1/Current actual value
//   Walking_Welding_Robot_Control_System/Walking_Welding_Robot_Control_System Instance <-> Device 3 (EtherCAT)/Drive 9 (Elmo Drive)
//     Simulink_Test Inputs/Walking_Robot_Control.Current_Turque_Value[9] <-> Inputs_1/Current actual value
//   Walking_Welding_Robot_Control_System/Walking_Welding_Robot_Control_System Instance <-> NC-Task 1 SAF/Axes/Axis 1
//     Simulink_Test Inputs/Walking_Robot_Control.Axis_Robot[1].AxisRef.NcToPlc <-> Outputs/ToPlc
//     Simulink_Test Outputs/Walking_Robot_Control.Axis_Robot[1].AxisRef.PlcToNc <-> Inputs/FromPlc
//   Walking_Welding_Robot_Control_System/Walking_Welding_Robot_Control_System Instance <-> NC-Task 1 SAF/Axes/Axis 10
//     Simulink_Test Inputs/Walking_Robot_Control.Axis_Robot[10].AxisRef.NcToPlc <-> Outputs/ToPlc
//     Simulink_Test Outputs/Walking_Robot_Control.Axis_Robot[10].AxisRef.PlcToNc <-> Inputs/FromPlc
//   Walking_Welding_Robot_Control_System/Walking_Welding_Robot_Control_System Instance <-> NC-Task 1 SAF/Axes/Axis 11
//     Simulink_Test Inputs/Walking_Robot_Control.Axis_Robot[11].AxisRef.NcToPlc <-> Outputs/ToPlc
//     Simulink_Test Outputs/Walking_Robot_Control.Axis_Robot[11].AxisRef.PlcToNc <-> Inputs/FromPlc
//   Walking_Welding_Robot_Control_System/Walking_Welding_Robot_Control_System Instance <-> NC-Task 1 SAF/Axes/Axis 12
//     Simulink_Test Inputs/Walking_Robot_Control.Axis_Robot[12].AxisRef.NcToPlc <-> Outputs/ToPlc
//     Simulink_Test Outputs/Walking_Robot_Control.Axis_Robot[12].AxisRef.PlcToNc <-> Inputs/FromPlc
//   Walking_Welding_Robot_Control_System/Walking_Welding_Robot_Control_System Instance <-> NC-Task 1 SAF/Axes/Axis 13
//     Simulink_Test Inputs/Walking_Robot_Control.Axis_Robot[13].AxisRef.NcToPlc <-> Outputs/ToPlc
//     Simulink_Test Outputs/Walking_Robot_Control.Axis_Robot[13].AxisRef.PlcToNc <-> Inputs/FromPlc
//   Walking_Welding_Robot_Control_System/Walking_Welding_Robot_Control_System Instance <-> NC-Task 1 SAF/Axes/Axis 14
//     Simulink_Test Inputs/Walking_Robot_Control.Axis_Robot[14].AxisRef.NcToPlc <-> Outputs/ToPlc
//     Simulink_Test Outputs/Walking_Robot_Control.Axis_Robot[14].AxisRef.PlcToNc <-> Inputs/FromPlc
//   Walking_Welding_Robot_Control_System/Walking_Welding_Robot_Control_System Instance <-> NC-Task 1 SAF/Axes/Axis 15
//     Simulink_Test Inputs/Walking_Robot_Control.Axis_Robot[15].AxisRef.NcToPlc <-> Outputs/ToPlc
//     Simulink_Test Outputs/Walking_Robot_Control.Axis_Robot[15].AxisRef.PlcToNc <-> Inputs/FromPlc
//   Walking_Welding_Robot_Control_System/Walking_Welding_Robot_Control_System Instance <-> NC-Task 1 SAF/Axes/Axis 16
//     Simulink_Test Inputs/Walking_Robot_Control.Axis_Robot[16].AxisRef.NcToPlc <-> Outputs/ToPlc
//     Simulink_Test Outputs/Walking_Robot_Control.Axis_Robot[16].AxisRef.PlcToNc <-> Inputs/FromPlc
//   Walking_Welding_Robot_Control_System/Walking_Welding_Robot_Control_System Instance <-> NC-Task 1 SAF/Axes/Axis 17
//     Simulink_Test Inputs/Walking_Robot_Control.Axis_Robot[17].AxisRef.NcToPlc <-> Outputs/ToPlc
//     Simulink_Test Outputs/Walking_Robot_Control.Axis_Robot[17].AxisRef.PlcToNc <-> Inputs/FromPlc
//   Walking_Welding_Robot_Control_System/Walking_Welding_Robot_Control_System Instance <-> NC-Task 1 SAF/Axes/Axis 18
//     Simulink_Test Inputs/Walking_Robot_Control.Axis_Robot[18].AxisRef.NcToPlc <-> Outputs/ToPlc
//     Simulink_Test Outputs/Walking_Robot_Control.Axis_Robot[18].AxisRef.PlcToNc <-> Inputs/FromPlc
//   Walking_Welding_Robot_Control_System/Walking_Welding_Robot_Control_System Instance <-> NC-Task 1 SAF/Axes/Axis 19
//     Simulink_Test Inputs/Welding_Arm_Control.Axis_Welding_Arm[1].AxisRef.NcToPlc <-> Outputs/ToPlc
//     Simulink_Test Outputs/Welding_Arm_Control.Axis_Welding_Arm[1].AxisRef.PlcToNc <-> Inputs/FromPlc
//   Walking_Welding_Robot_Control_System/Walking_Welding_Robot_Control_System Instance <-> NC-Task 1 SAF/Axes/Axis 2
//     Simulink_Test Inputs/Walking_Robot_Control.Axis_Robot[2].AxisRef.NcToPlc <-> Outputs/ToPlc
//     Simulink_Test Outputs/Walking_Robot_Control.Axis_Robot[2].AxisRef.PlcToNc <-> Inputs/FromPlc
//   Walking_Welding_Robot_Control_System/Walking_Welding_Robot_Control_System Instance <-> NC-Task 1 SAF/Axes/Axis 20
//     Simulink_Test Inputs/Welding_Arm_Control.Axis_Welding_Arm[2].AxisRef.NcToPlc <-> Outputs/ToPlc
//     Simulink_Test Outputs/Welding_Arm_Control.Axis_Welding_Arm[2].AxisRef.PlcToNc <-> Inputs/FromPlc
//   Walking_Welding_Robot_Control_System/Walking_Welding_Robot_Control_System Instance <-> NC-Task 1 SAF/Axes/Axis 21
//     Simulink_Test Inputs/Welding_Arm_Control.Axis_Welding_Arm[3].AxisRef.NcToPlc <-> Outputs/ToPlc
//     Simulink_Test Outputs/Welding_Arm_Control.Axis_Welding_Arm[3].AxisRef.PlcToNc <-> Inputs/FromPlc
//   Walking_Welding_Robot_Control_System/Walking_Welding_Robot_Control_System Instance <-> NC-Task 1 SAF/Axes/Axis 22
//     Simulink_Test Inputs/Welding_Arm_Control.Axis_Welding_Arm[4].AxisRef.NcToPlc <-> Outputs/ToPlc
//     Simulink_Test Outputs/Welding_Arm_Control.Axis_Welding_Arm[4].AxisRef.PlcToNc <-> Inputs/FromPlc
//   Walking_Welding_Robot_Control_System/Walking_Welding_Robot_Control_System Instance <-> NC-Task 1 SAF/Axes/Axis 23
//     Simulink_Test Inputs/Welding_Arm_Control.Axis_Welding_Arm[5].AxisRef.NcToPlc <-> Outputs/ToPlc
//     Simulink_Test Outputs/Welding_Arm_Control.Axis_Welding_Arm[5].AxisRef.PlcToNc <-> Inputs/FromPlc
//   Walking_Welding_Robot_Control_System/Walking_Welding_Robot_Control_System Instance <-> NC-Task 1 SAF/Axes/Axis 24
//     Simulink_Test Inputs/Welding_Arm_Control.Axis_Welding_Arm[6].AxisRef.NcToPlc <-> Outputs/ToPlc
//     Simulink_Test Outputs/Welding_Arm_Control.Axis_Welding_Arm[6].AxisRef.PlcToNc <-> Inputs/FromPlc
//   Walking_Welding_Robot_Control_System/Walking_Welding_Robot_Control_System Instance <-> NC-Task 1 SAF/Axes/Axis 3
//     Simulink_Test Inputs/Walking_Robot_Control.Axis_Robot[3].AxisRef.NcToPlc <-> Outputs/ToPlc
//     Simulink_Test Outputs/Walking_Robot_Control.Axis_Robot[3].AxisRef.PlcToNc <-> Inputs/FromPlc
//   Walking_Welding_Robot_Control_System/Walking_Welding_Robot_Control_System Instance <-> NC-Task 1 SAF/Axes/Axis 4
//     Simulink_Test Inputs/Walking_Robot_Control.Axis_Robot[4].AxisRef.NcToPlc <-> Outputs/ToPlc
//     Simulink_Test Outputs/Walking_Robot_Control.Axis_Robot[4].AxisRef.PlcToNc <-> Inputs/FromPlc
//   Walking_Welding_Robot_Control_System/Walking_Welding_Robot_Control_System Instance <-> NC-Task 1 SAF/Axes/Axis 5
//     Simulink_Test Inputs/Walking_Robot_Control.Axis_Robot[5].AxisRef.NcToPlc <-> Outputs/ToPlc
//     Simulink_Test Outputs/Walking_Robot_Control.Axis_Robot[5].AxisRef.PlcToNc <-> Inputs/FromPlc
//   Walking_Welding_Robot_Control_System/Walking_Welding_Robot_Control_System Instance <-> NC-Task 1 SAF/Axes/Axis 6
//     Simulink_Test Inputs/Walking_Robot_Control.Axis_Robot[6].AxisRef.NcToPlc <-> Outputs/ToPlc
//     Simulink_Test Outputs/Walking_Robot_Control.Axis_Robot[6].AxisRef.PlcToNc <-> Inputs/FromPlc
//   Walking_Welding_Robot_Control_System/Walking_Welding_Robot_Control_System Instance <-> NC-Task 1 SAF/Axes/Axis 7
//     Simulink_Test Inputs/Walking_Robot_Control.Axis_Robot[7].AxisRef.NcToPlc <-> Outputs/ToPlc
//     Simulink_Test Outputs/Walking_Robot_Control.Axis_Robot[7].AxisRef.PlcToNc <-> Inputs/FromPlc
//   Walking_Welding_Robot_Control_System/Walking_Welding_Robot_Control_System Instance <-> NC-Task 1 SAF/Axes/Axis 8
//     Simulink_Test Inputs/Walking_Robot_Control.Axis_Robot[8].AxisRef.NcToPlc <-> Outputs/ToPlc
//     Simulink_Test Outputs/Walking_Robot_Control.Axis_Robot[8].AxisRef.PlcToNc <-> Inputs/FromPlc
//   Walking_Welding_Robot_Control_System/Walking_Welding_Robot_Control_System Instance <-> NC-Task 1 SAF/Axes/Axis 9
//     Simulink_Test Inputs/Walking_Robot_Control.Axis_Robot[9].AxisRef.NcToPlc <-> Outputs/ToPlc
//     Simulink_Test Outputs/Walking_Robot_Control.Axis_Robot[9].AxisRef.PlcToNc <-> Inputs/FromPlc

CONFIGURATION Walking_Welding_Robot_Control_System
    RESOURCE PLC ON TwinCAT3
        TASK PlcTask(INTERVAL := T#4ms, PRIORITY := 12);
        TASK Sensor_Test(INTERVAL := T#1ms, PRIORITY := 14);
        TASK Simulink_Test(INTERVAL := T#4ms, PRIORITY := 6);
        PROGRAM Walking_Robot_Control WITH PlcTask : Walking_Robot_Control;
        PROGRAM Welding_Arm_Control WITH PlcTask : Welding_Arm_Control;
        PROGRAM Walking_Welding_Robot_Control WITH PlcTask : Walking_Welding_Robot_Control;
        PROGRAM SignalData_Interface WITH Sensor_Test : SignalData_Interface;
        PROGRAM Walking_Robot_Movement WITH Simulink_Test : Walking_Robot_Movement;
        PROGRAM Welding_Arm_Movement WITH Simulink_Test : Welding_Arm_Movement;
    END_RESOURCE
END_CONFIGURATION

// ---- DUTs/Filter_Current/ST_Filter_Current_Hexapod_Robot_InitData.TcDUT
{attribute 'pack_mode' := '4'}
TYPE ST_Filter_Current_Hexapod_Robot_InitData :
STRUCT
	Header: TComInitDataHdr;
	CallByHdr: TComInitDataElmHdr;
	CallBy: TctModuleCallByType;
	ExecutionSequenceHdr: TComInitDataElmHdr;
	ExecutionSequence: TctModuleExecutionSequenceType;
	StepSizeHdr: TComInitDataElmHdr;
	StepSize: TctStepSizeType;
	ExecuteModelCodeHdr: TComInitDataElmHdr;
	ExecuteModelCode: BOOL;
	ModelParametersHdr: TComInitDataElmHdr;
	ModelParameters: P_Filter_Current_Hexapod_Robo_T;
	ContextInfoArr_0_TaskOidHdr: TComInitDataElmHdr;
	ContextInfoArr_0_TaskOid: OTCID;
	ContextInfoArr_0_TaskPriorityHdr: TComInitDataElmHdr;
	ContextInfoArr_0_TaskPriority: UDINT;
	ContextInfoArr_0_TaskCycleTimeNsHdr: TComInitDataElmHdr;
	ContextInfoArr_0_TaskCycleTimeNs: UDINT;
	ContextInfoArr_0_TaskPortHdr: TComInitDataElmHdr;
	ContextInfoArr_0_TaskPort: UINT;
	ContextInfoArr_0_TaskSortOrderHdr: TComInitDataElmHdr;
	ContextInfoArr_0_TaskSortOrder: UDINT;
END_STRUCT
END_TYPE

// ---- DUTs/Filter_Current/ST_Filter_Current_Hexapod_Robot_Input.TcDUT
TYPE ST_Filter_Current_Hexapod_Robot_Input :
STRUCT
	Current_Motor: matrix_18_real_T;
END_STRUCT
END_TYPE

// ---- DUTs/Filter_Current/ST_Filter_Current_Hexapod_Robot_Output.TcDUT
TYPE ST_Filter_Current_Hexapod_Robot_Output :
STRUCT
	Current_Monitor: matrix_18_real_T;
END_STRUCT
END_TYPE

// ---- DUTs/Touch_Signal_Detection/ST_Tough_Signal_Detection_Simple_InitData.TcDUT
{attribute 'pack_mode' := '4'}
TYPE ST_Tough_Signal_Detection_Simple_InitData :
STRUCT
	Header: TComInitDataHdr;
	CallByHdr: TComInitDataElmHdr;
	CallBy: TctModuleCallByType;
	ExecutionSequenceHdr: TComInitDataElmHdr;
	ExecutionSequence: TctModuleExecutionSequenceType;
	StepSizeHdr: TComInitDataElmHdr;
	StepSize: TctStepSizeType;
	ExecuteModelCodeHdr: TComInitDataElmHdr;
	ExecuteModelCode: BOOL;
	ModelParametersHdr: TComInitDataElmHdr;
	ModelParameters: P_Touch_Signal_Detection_Simp_T;
	ContextInfoArr_0_TaskOidHdr: TComInitDataElmHdr;
	ContextInfoArr_0_TaskOid: OTCID;
	ContextInfoArr_0_TaskPriorityHdr: TComInitDataElmHdr;
	ContextInfoArr_0_TaskPriority: UDINT;
	ContextInfoArr_0_TaskCycleTimeNsHdr: TComInitDataElmHdr;
	ContextInfoArr_0_TaskCycleTimeNs: UDINT;
	ContextInfoArr_0_TaskPortHdr: TComInitDataElmHdr;
	ContextInfoArr_0_TaskPort: UINT;
	ContextInfoArr_0_TaskSortOrderHdr: TComInitDataElmHdr;
	ContextInfoArr_0_TaskSortOrder: UDINT;
END_STRUCT
END_TYPE

// ---- DUTs/Touch_Signal_Detection/ST_Tough_Signal_Detection_Simple_Input.TcDUT
TYPE ST_Tough_Signal_Detection_Simple_Input :
STRUCT
	Current_Filter: matrix_18_real_T;
	Delay_Time: LREAL;
	Minimum_Limit: LREAL;
	State: LREAL;
	Number: LREAL;
END_STRUCT
END_TYPE

// ---- DUTs/Touch_Signal_Detection/ST_Tough_Signal_Detection_Simple_Output.TcDUT
TYPE ST_Tough_Signal_Detection_Simple_Output :
STRUCT
	Touch_Signal: matrix_6_boolean_T;
	Leg_Touch: matrix_3_real_T;
	Leg_Detection: matrix_3_real_T;
	Current_Change: matrix_18_real_T;
END_STRUCT
END_TYPE

// ---- DUTs/Welding_Arm_Simulink/ST_WeldingArm6AxisMotion_Control_InitData.TcDUT
{attribute 'pack_mode' := '4'}
TYPE ST_WeldingArm6AxisMotion_Control_InitData :
STRUCT
	Header: TComInitDataHdr;
	CallByHdr: TComInitDataElmHdr;
	CallBy: TctModuleCallByType;
	ExecutionSequenceHdr: TComInitDataElmHdr;
	ExecutionSequence: TctModuleExecutionSequenceType;
	StepSizeHdr: TComInitDataElmHdr;
	StepSize: TctStepSizeType;
	ExecuteModelCodeHdr: TComInitDataElmHdr;
	ExecuteModelCode: BOOL;
	ModelParametersHdr: TComInitDataElmHdr;
	ModelParameters: P_weldingArm6axisMotionTest1_T;
	ContextInfoArr_0_TaskOidHdr: TComInitDataElmHdr;
	ContextInfoArr_0_TaskOid: OTCID;
	ContextInfoArr_0_TaskPriorityHdr: TComInitDataElmHdr;
	ContextInfoArr_0_TaskPriority: UDINT;
	ContextInfoArr_0_TaskCycleTimeNsHdr: TComInitDataElmHdr;
	ContextInfoArr_0_TaskCycleTimeNs: UDINT;
	ContextInfoArr_0_TaskPortHdr: TComInitDataElmHdr;
	ContextInfoArr_0_TaskPort: UINT;
	ContextInfoArr_0_TaskSortOrderHdr: TComInitDataElmHdr;
	ContextInfoArr_0_TaskSortOrder: UDINT;
END_STRUCT
END_TYPE

// ---- DUTs/Welding_Arm_Simulink/ST_WeldingArm6AxisMotion_Control_Input.TcDUT
TYPE ST_WeldingArm6AxisMotion_Control_Input :
STRUCT
	t: LREAL;
END_STRUCT
END_TYPE

// ---- DUTs/Welding_Arm_Simulink/ST_WeldingArm6AxisMotion_Control_Output.TcDUT
TYPE ST_WeldingArm6AxisMotion_Control_Output :
STRUCT
	Disp_J: matrix_6_real_T;
	T_ALL: LREAL;
END_STRUCT
END_TYPE

// ---- POUs/Walking_Robot_Control.TcPOU
PROGRAM Walking_Robot_Control
VAR_INPUT
	// ====== 模块动作信号(按动作先后排列) ======
	Power_Execute 			: BOOL;							// 上电使能
	Axis_Power				: ARRAY[1..18] OF BOOL;		// 单电机上电
	Robot_Power				: BOOL;							// 所有电机同时上电
	
	Home_Execute			: BOOL;							// 找零使能
	Leg_Home_Set			: ARRAY[1..6] OF BOOL;			// 单腿找零
	Axis_Home_Set			: ARRAY[1..18] OF BOOL;		// 单电机找零
	Robot_Home_Set			: BOOL;							// 所有电机同时找零
	
	Reset_Execute			: BOOL;							// 重置使能
	Axis_Reset				: ARRAY[1..18] OF BOOL;		// 单电机重置
	Robot_Reset				: BOOL;							// 所有电机同时重置
	
	Move_Execute			: BOOL;							// 绝对运动使能
	Robot_Stand_Execute		: BOOL;							// 机器人站立程序使能	
	Axis_Absolute_Eable		: ARRAY[1..18] OF BOOL;		// 单电机绝对运动
	Axis_Move_Position		: ARRAY[1..18] OF LREAL;		// 单电机绝对运动位置			
END_VAR

VAR
	// ====== NC轴变量 ======
	Axis_Robot				: ARRAY[1..18] OF Axis;			// 定义六足轴参量(可以调整数据上限来调整电机数目)
	Leg_Number				: INT;							// 定义六足腿数量
	Axis_Number 			: INT;							// 定义留住轴数量
	
	// ====== 状态监测变量 ======
	Power_Status			: ARRAY[1..18] OF BOOL;		// 单电机上电状态
	Robot_Home_Done			: BOOL;							// 六足机器人找零完成信号
	Tripod_Home_Done		: ARRAY[1..2] OF BOOL;			// 单组腿(一组三条,134或246)找零完成信号
	Leg_Home_Done			: ARRAY[1..6] OF BOOL;			// 单条腿找零完成信号
	Home_Done				: ARRAY[1..18] OF BOOL;		// 单电机找零完成信号
	MoveAbsoluteDone		: ARRAY[1..18] OF BOOL;		// 单电机运动监测信号
	
	Robot_Error				: BOOL;							// 机器人错误信号
	Axis_Error				: ARRAY[1..18] OF BOOL;		// 单电机错误信号
	Axis_ErrorID			: ARRAY[1..18] OF UDINT;		// 单电机错误码
	
	Axis_ActPostion			: ARRAY[1..18] OF LREAL;		// 单电机轴实际位置
	Axis_ActVelocity		: ARRAY[1..18] OF LREAL;		// 单电机轴实际速度
	
	// ====== Simulink模型与控制模型映射 ======
	// 需要注意映射前后分别代表什么
	Mapping_ActPosition		: Variable_Control_Mapping_Model;// 电机位置映射
	Motor_ActPosition		: ARRAY[1..18] OF LREAL;		// Mapping后的电机轴实际位置
	
	Max_Turque_Value		: INT;							// 设置最大力矩边界值
	
	Mapping_Current			: Variable_Control_Mapping_Model;// 电流值映射
	Current_Turque_Value AT%IW0 : ARRAY[1..18] OF INT;		// 驱动检测到的实际电机的力矩
	Current_Before_Mapping	: ARRAY[1..18] OF LREAL ;		// 将Current_Turque_Value从INT转换成LREAL,用来进行变量监测
	Current_After_Mapping	: ARRAY[1..18] OF LREAL;		// 映射后的电流值,即Simulink对应腿的电流
END_VAR


Variable_Monitor();				// 变量监测程序

Logic_Control();				// 逻辑控制程序

Variable_Set();					// 变量设定程序

Leg_Action();					// 单腿运动程序

Robot_Action();					// 机器人整体运动程序

Robot_Single_Motor_Action();	// 机器人单个电机运动程序

ACTION Leg_Action:

// ====== 机器人单挑腿找零程序 ======
IF Home_Execute THEN
	FOR Leg_Number := 1 TO 6 {BY 1} DO
		IF Leg_Home_Set[Leg_Number] THEN
			// 某条腿找零,即代表该条腿上的三个电机就开始找零
			Axis_Home_Set[1+(Leg_Number-1)*3] := Leg_Home_Set[Leg_Number];
			Axis_Home_Set[2+(Leg_Number-1)*3] := Leg_Home_Set[Leg_Number];
			Axis_Home_Set[3+(Leg_Number-1)*3] := Leg_Home_Set[Leg_Number];
		ELSIF Home_Done[1+(Leg_Number-1)*3] AND Home_Done[2+(Leg_Number-1)*3] AND Home_Done[3+(Leg_Number-1)*3] THEN
			// 某条腿上三个电机找零结束,[单腿找零]信号关闭
			// 实际上,这个ELSIF不可能进入,因为Home_Done是一个宽度为PLC周期的脉冲信号,一腿上三个电机不可能同时找零完成
			// 在Logic_Control中规定了Home_Done信号发生即对Axis_Home_Set置FALSE,因此不用担心找零完成后[单电机找零]还处于开启状态
			Leg_Home_Set[Leg_Number] := FALSE; 
			Axis_Home_Set[1+(Leg_Number-1)*3] := FALSE;
			Axis_Home_Set[2+(Leg_Number-1)*3] := FALSE;
			Axis_Home_Set[3+(Leg_Number-1)*3] := FALSE;
		END_IF
					
		// 由于Home_Done信号不会同时发生,因此不能用它来判断是否单腿找零完成(单腿三电机都找零完成),可以适用位置来判断
		// Simulink模型规定的单腿三电机初始位置与实际位置误差均小于0.01后,即可认为单腿找零完成
		// 这里的Walking_Robot_Movement.Mapping_Position.Controller_Leg_Variable也可使用Axis_Robot[Axis_Number].Home_Absolute_Position
		// 因为已经在Variable_Set中将前者设定为后者了
		IF ABS(Walking_Robot_Movement.Mapping_Position.Controller_Leg_Variable[1+(Leg_Number-1)*3]-Axis_ActPostion[1+(Leg_Number-1)*3])<0.1 AND 
			ABS(Walking_Robot_Movement.Mapping_Position.Controller_Leg_Variable[2+(Leg_Number-1)*3]-Axis_ActPostion[2+(Leg_Number-1)*3])<0.1 AND
			ABS(Walking_Robot_Movement.Mapping_Position.Controller_Leg_Variable[3+(Leg_Number-1)*3]-Axis_ActPostion[3+(Leg_Number-1)*3])<0.1 THEN
			Leg_Home_Done[Leg_Number]	:= TRUE;
		ELSE
			Leg_Home_Done[Leg_Number]	:= FALSE;
		END_IF

		// 单组三腿135均完成找零,则该组腿找零完成
		IF Leg_Home_Done[1] AND Leg_Home_Done[3] AND Leg_Home_Done[5] THEN
			Tripod_Home_Done[1]		:= TRUE;
		ELSE
			Tripod_Home_Done[1]		:= FALSE;
		END_IF
		// 单组三腿246均完成找零,则该组腿找零完成
		IF Leg_Home_Done[2] AND Leg_Home_Done[4] AND Leg_Home_Done[6] THEN
			Tripod_Home_Done[2]		:= TRUE;
		ELSE
			Tripod_Home_Done[2]		:= FALSE;
		END_IF
		
		// 两组都找零完成,则整个机器人找零完成
		IF Tripod_Home_Done[1]	AND Tripod_Home_Done[2]	THEN
			Robot_Home_Done			:= TRUE;
		ELSE
			Robot_Home_Done			:= FALSE;
		END_IF
	END_FOR
ELSIF NOT Home_Execute THEN
	Robot_Home_Done 	:= FALSE;
	Tripod_Home_Done[1] := FALSE;
	Tripod_Home_Done[2] := FALSE;
	FOR Leg_Number := 1 TO 6 {BY 1} DO
		Leg_Home_Done[Leg_Number] := FALSE;
	END_FOR
END_IF

// ====== 机器人其它单腿运动程序 ======
END_ACTION

ACTION Logic_Control:
// =======================控制逻辑区==========================
// 保证所有的动作拥有合理的先后顺序，优化控制逻辑
// 也防止出现两个或两个以上动作同时进行的情况，保证控制安全

// ====== 电机驱动重置逻辑 ======
IF Axis_Error[1] OR Axis_Error[2] OR Axis_Error[3] OR Axis_Error[4] OR Axis_Error[5] OR Axis_Error[6]
	 OR Axis_Error[7] OR Axis_Error[8] OR Axis_Error[9] OR Axis_Error[10] OR Axis_Error[11] OR Axis_Error[12]
		OR Axis_Error[13] OR Axis_Error[14] OR Axis_Error[15] OR Axis_Error[16] OR Axis_Error[17] OR Axis_Error[18] THEN
	// 某一个电机出现错误,代表整个六足即有错
	Robot_Error := TRUE;
ELSE
	Robot_Error := FALSE;
END_IF

IF Robot_Error THEN
	// 电机出现错误,则[驱动重置]开关开启,允许重置
	Reset_Execute := TRUE;
ELSIF NOT Robot_Error THEN
	// 电机没有错误,则[驱动重置]开关关闭,不允许重置
	Reset_Execute := FALSE;
END_IF

	// [重置使能]关闭,所有电机均不能重置
IF NOT Reset_Execute THEN
	FOR Axis_Number := 1 TO 18 {BY 1} DO
		Axis_Reset[Axis_Number] := FALSE;
		Axis_Robot[Axis_Number].Reset(Drive_Reset:= Axis_Reset[Axis_Number]);
	END_FOR
END_IF

	// 这五行两个作用： 1. 若电机没错误,则不允许重置
	// 2. 清除错误后自动将[单电机重置]信号关闭,不然得手动关闭
FOR Axis_Number := 1 TO 18 {BY 1} DO
	IF NOT Axis_Error[Axis_Number] THEN
		Axis_Reset[Axis_Number] := FALSE;
	END_IF
END_FOR

// ====== 上电程序逻辑 ======
IF NOT Power_Execute THEN
	// [上电使能]关闭,所有电机必须立即断电
	FOR Axis_Number := 1 TO 18 {BY 1} DO
		Axis_Power[Axis_Number] := FALSE;
		Axis_Robot[Axis_Number].Power(Axis_Enable:= Axis_Power[Axis_Number]);
	END_FOR
	// 未上电时，不能进行找零
	Home_Execute := FALSE;			
	// 未上电时，不能进行运动
	Move_Execute := FALSE;			
END_IF

// ====== 找零程序逻辑 ======
IF Home_Execute THEN
	FOR Axis_Number := 1 TO 18 {BY 1} DO
		// 	丝杠到达零点位置后，单电机标零使能位关闭		
		IF Home_Done[Axis_Number] THEN				
			Axis_Home_Set[Axis_Number] :=0;	
			Axis_Robot[Axis_Number].Home(Drive_Home:= Axis_Home_Set[Axis_Number]);
		END_IF
	END_FOR
	// 设定零点时，不能进行运动
	Move_Execute :=0;							
ELSIF NOT Home_Execute THEN
	// [找零使能]关闭,不允许找零
	FOR Axis_Number := 1 TO 18 {BY 1} DO
		Axis_Home_Set[Axis_Number] := 0;
	END_FOR
END_IF

// ====== 机器人站立逻辑 ======
IF Move_Execute THEN
	// 站立运动使能时，机器人调零必须结束
	Home_Execute := FALSE;
	FOR Axis_Number := 1 TO 18 {BY 1} DO
		// 	丝杠到达设定位置后，单电机绝对运动使能位关闭
		IF MoveAbsoluteDone[Axis_Number] THEN	
			Axis_Absolute_Eable[Axis_Number] := FALSE;
		END_IF
	END_FOR
ELSIF NOT Move_Execute THEN						
	// 站立运动不使能,轴不能运动
	FOR Axis_Number := 1 TO 18 {BY 1} DO
		Axis_Absolute_Eable[Axis_Number] := FALSE;
		Axis_Robot[Axis_Number].Move_Absolute(	Drive_Move_Absolute:= Axis_Absolute_Eable[Axis_Number], 
												Absolute_Position:= Axis_Move_Position[Axis_Number]);
	END_FOR
END_IF
END_ACTION

ACTION Robot_Action:
// =================机器人整体运动命令区======================
// 六足所有电机整体控制

// ====== 机器人所有驱动同时重置 ======
IF Robot_Reset THEN
	// [重置使能]前提下,才能重置
	IF Reset_Execute THEN
		FOR Axis_Number := 1 TO 18 {BY 1} DO
			Axis_Reset[Axis_Number] := TRUE;
			Axis_Robot[Axis_Number].Reset(Drive_Reset:= Axis_Reset[Axis_Number]);
		END_FOR
	END_IF
END_IF	

// ====== 机器人所有电机同时上电 ======
IF Robot_Power THEN	
	// [上电使能]前提下,才能上电
	IF Power_Execute THEN
		FOR Axis_Number := 1 TO 18 {BY 1} DO
			Axis_Power[Axis_Number] := TRUE ;
			Axis_Robot[Axis_Number].Power(Axis_Enable:= Axis_Power[Axis_Number]);
		END_FOR
	END_IF
END_IF
	
// ====== 机器人所有电机同时找零 ======
IF Robot_Home_Set THEN
	IF Home_Execute THEN
		// 在整机调零时,1\3\5三条腿或者2\4\6三条腿同时找零,由于总需要3条腿触地支撑,因此不能6条腿同时找零
		// 因此,某组腿找零,另一组不允许找零. (机器人吊起时,六腿离地,可以6腿找零,但为了安全不考虑该情况)
		IF Leg_Home_Set[1] THEN
			Leg_Home_Set[2] := FALSE;
		END_IF
		IF Leg_Home_Set[2] THEN
			Leg_Home_Set[1] := FALSE;
		END_IF
		// 只有按腿1或者腿2可以同时进行三条腿找零,因为三条腿不可能在同一个PLC内同时完成找零
		Leg_Home_Set[3] := Leg_Home_Set[5] := Leg_Home_Set[1];
		Leg_Home_Set[4] := Leg_Home_Set[6] := Leg_Home_Set[2];
	ELSIF NOT Home_Execute THEN
		// [找零使能]关闭,不允许找零
		FOR Leg_Number := 1 TO 6 {BY 1} DO
			Leg_Home_Set[Leg_Number] := FALSE;
		END_FOR
	END_IF
ELSIF NOT Robot_Home_Set AND NOT Home_Execute THEN
	FOR Axis_Number := 1 TO 18 {BY 1} DO
		Axis_Home_Set[Axis_Number] := FALSE;
	END_FOR
END_IF

// ====== 机器人站立,用于Visu_Walking_Robot_Stand调试 ======
IF Robot_Stand_Execute THEN
	IF Move_Execute THEN
		FOR Axis_Number := 1 TO 18 {BY 1} DO
			// 丝杠到达设定位置后，单电机绝对运动使能位关闭
			IF MoveAbsoluteDone[Axis_Number] THEN		
				Axis_Absolute_Eable[Axis_Number] := FALSE;
			ELSE
				Axis_Absolute_Eable[Axis_Number] := TRUE;
			END_IF
		END_FOR
	END_IF
ELSIF NOT Robot_Stand_Execute AND NOT Move_Execute THEN 
	FOR Axis_Number := 1 TO 18 {BY 1} DO
		Axis_Absolute_Eable[Axis_Number] := FALSE;
	END_FOR
END_IF
END_ACTION

ACTION Robot_Single_Motor_Action:

// ====== 单电机驱动重置 ======
IF Reset_Execute THEN
	FOR Axis_Number := 1 TO 18 {BY 1} DO
		Axis_Robot[Axis_Number].Reset(Drive_Reset:= Axis_Reset[Axis_Number]);
	END_FOR
END_IF

// ====== 单电机上电 ======
IF Power_Execute THEN
	FOR Axis_Number := 1 TO 18 {BY 1} DO
		Axis_Robot[Axis_Number].Power(Axis_Enable:= Axis_Power[Axis_Number]);
	END_FOR
END_IF

// ====== 单电机找零 ======
IF Home_Execute THEN
	FOR Axis_Number := 1 TO 18 {BY 1} DO
		Axis_Robot[Axis_Number].Home(Drive_Home:= Axis_Home_Set[Axis_Number]);
	END_FOR
END_IF

// ====== 单电机站立 ======
IF Move_Execute THEN
	FOR Axis_Number := 1 TO 18 {BY 1} DO
		Axis_Robot[Axis_Number].Move_Absolute(	Drive_Move_Absolute:= Axis_Absolute_Eable[Axis_Number], 
												Absolute_Position:= Axis_Move_Position[Axis_Number]);
	END_FOR
END_IF
END_ACTION

ACTION Safety:
// 保证丝杠行程和电机速度在规定范围内
END_ACTION

ACTION Variable_Monitor:
// =====================关键数据信号监测======================

// ====== 设置最大力矩(边界控制条件) ======
FOR Axis_Number := 1 TO 18 {BY 1} DO
	Axis_Robot[Axis_Number].Max_Turque_Value := Max_Turque_Value;
END_FOR

// ====== 检测、映射力矩 ======
FOR Axis_Number := 1 TO 18 {BY 1} DO
	// 检测实际力矩,Current_Turque_Value 链接到I/O中对应电机的Digital_Input_1(即驱动监测到的实际力矩)
	Axis_Robot[Axis_Number].Current_Turque_Value := Current_Turque_Value[Axis_Number];
	// 驱动监测到的实际力矩为INT,而Mapping_Current的输入,输出均是LREAL,需要进行变量强制转换
	Current_Before_Mapping[Axis_Number] := INT_TO_LREAL(Current_Turque_Value[Axis_Number]);
END_FOR
	// 将检测到的电机实际力矩,映射到Simulink控制模型中对应腿的力矩
Mapping_Current(Controller_Leg_Variable:= Current_Before_Mapping, Model_Leg_Variable=> Current_After_Mapping);

// ====== 检测轴实际位置、速度检测区 ======
FOR Axis_Number := 1 TO 18 {BY 1} DO
	Axis_ActPostion[Axis_Number] := Axis_Robot[Axis_Number].ActPosition;
	Axis_ActVelocity[Axis_Number] := Axis_Robot[Axis_Number].ActVelocity;
END_FOR
	// 将检测到的电机实际位置,映射到Simulink控制模型中对应腿的位置
Mapping_ActPosition(Controller_Leg_Variable:= Axis_ActPostion, Model_Leg_Variable=> Motor_ActPosition);

// ====== 检测上电状态 ======
FOR Axis_Number := 1 TO 18 {BY 1} DO
	Power_Status[Axis_Number] := Axis_Robot[Axis_Number].State_PowerStatus;
END_FOR

// ====== 检测找零状态 ======
FOR Axis_Number := 1 TO 18 {BY 1} DO
	Home_Done[Axis_Number] := Axis_Robot[Axis_Number].State_HomeDone;
END_FOR

// ====== 检测绝对运动状态 ======
FOR Axis_Number := 1 TO 18 {BY 1} DO
	MoveAbsoluteDone[Axis_Number] := Axis_Robot[Axis_Number].State_MoveAbsoluteDone;
END_FOR

// ====== 检测电机错误 ======
FOR Axis_Number := 1 TO 18 {BY 1} DO
	Axis_Error[Axis_Number] := Axis_Robot[Axis_Number].Axis_Error;
	Axis_ErrorID[Axis_Number] := Axis_Robot[Axis_Number].Axis_ErrorID;
END_FOR
END_ACTION

ACTION Variable_Set:
// 注意：找零有两个过程
//		1. 丝杠回退到顶点,设置该处为零点  
//		2. 设完零点后运动到Simulink模型中各电机的初始位置(一般不为零)

// ====== 设定速度 ======
FOR Axis_Number := 1 TO 18 {BY 1} DO
	// 设定每个轴找零时过程1的速度
	Axis_Robot[Axis_Number].Home_Velocity 	:= 20;
	// 设定每个轴进行相对运动的速度
	Axis_Robot[Axis_Number].Move_Relative_Velocity	:=30;
END_FOR

IF Home_Execute THEN
	// 设定每各轴找零时过程2的速度,此速度可以保证每个轴不会在地面拖拽
	Axis_Robot[1].Move_Absolute_Velocity :=17;
	Axis_Robot[3].Move_Absolute_Velocity :=17; 
	Axis_Robot[4].Move_Absolute_Velocity :=16.74;
	Axis_Robot[6].Move_Absolute_Velocity :=16.74; 
	Axis_Robot[7].Move_Absolute_Velocity :=17.3; 
	Axis_Robot[9].Move_Absolute_Velocity :=17.3;
	Axis_Robot[10].Move_Absolute_Velocity :=16.95; 
	Axis_Robot[12].Move_Absolute_Velocity :=16.95; 
	Axis_Robot[13].Move_Absolute_Velocity :=17;
	Axis_Robot[15].Move_Absolute_Velocity :=17; 
	Axis_Robot[16].Move_Absolute_Velocity :=17; 
	Axis_Robot[18].Move_Absolute_Velocity :=17;
	Axis_Robot[2].Move_Absolute_Velocity :=20; 
	Axis_Robot[5].Move_Absolute_Velocity :=19.8; 
	Axis_Robot[8].Move_Absolute_Velocity :=20;
	Axis_Robot[11].Move_Absolute_Velocity :=20; 
	Axis_Robot[14].Move_Absolute_Velocity :=20; 
	Axis_Robot[17].Move_Absolute_Velocity :=20;
ELSE
	FOR Axis_Number := 1 TO 18 {BY 1} DO
		// 如果不处在找零时,则绝对运动速度设一个较小值,保证安全
		Axis_Robot[Axis_Number].Move_Absolute_Velocity	:=10;
	END_FOR
END_IF

// ====== 规定绝对运动位置 ======
	// 每次进行绝对位置都运动到160mm处
FOR Axis_Number := 1 TO 18 {BY 1} DO
	Axis_Move_Position[Axis_Number] := 160;
END_FOR

// ====== 规定最大力矩 ======
	// 此力矩用于判定在找零时过程1是否丝杠顶到了顶点
	// 该值不宜过大或过小,过大会损坏丝杠,过小会使找零过程2使脚触地后被判断为顶到了顶点
	// 经测试可以设置为1400,找零过程2脚触底的力矩值约在1000出头
Max_Turque_Value := 1400;

// ====== 设定电机找零时过程2的Simulink初始位置 =======
IF Home_Execute THEN
	FOR Axis_Number := 1 TO 18 {BY 1} DO
		Axis_Robot[Axis_Number].Home_Absolute_Position := Walking_Robot_Movement.Mapping_Position.Controller_Leg_Variable[Axis_Number];
	END_FOR
END_IF
END_ACTION

END_PROGRAM

// ---- DUTs/Axis/Axis.TcPOU
FUNCTION_BLOCK Axis
//VAR_INPUT	
//END_VAR
VAR_OUTPUT
	Axis_Error			: BOOL;				// Error signal
	Axis_ErrorID		: UDINT;			// Error ID
	Axis_Moves			: BOOL;				// Status of moving
END_VAR
VAR
	// =============== Done signals MC Block =================
	JogDone			    : BOOL;					// Status of function block MC_Jog
	ResetDone		    : BOOL;					// Status of function block MC_Reset
	HaltDone		    : BOOL;					// Status of function block MC_Halt
	HomeDone		    : BOOL;					// Status of function block MC_Home
  	MoveAbsoluteDone : BOOL;        // Status of function block MC_MoveAbsolute
    MoveRelativeDone  : BOOL;     // Status of function block MC_MoveRelative
  	ExtSetPiontDone 	: BOOL;         		// Status of function block MC_ExtSetPointGenDisable

	// =============== Control variables ======================
	//Home_Back_Start	: BOOL;
	//Drive_Home		: BOOL;
	
	// =============== State variables ========================
	Power_StatusEnable	: BOOL;					// Enable feedback
	
	// ============= Velocity, override ,Position==============
	Velocity_Jog		: LREAL;				// Jog velocity
	Velocity_Move		: LREAL;				// Target velocity
	Velocity_Home		: LREAL;				// Home velocity
	Velocity_Absolute	: LREAL;				// MoveAbsolute velocity
	Velocity_Relative	: LREAL;				// MoveRelative velocity
	fOverride 			: LREAL := 100.0;		// Override 100%
  	Home_Position   : LREAL;        // The absolute position after Home will be
	
	// =============== Trigger function blocks ================
	
	TriggerHalt	: R_TRIG;				// Trigger to recognize rising edge of halt input
	TriggerReset : R_TRIG;				// Trigger to recognize rising edge of reset input
	
	// =============== Axis reference =========================
	AxisRef			: AXIS_REF;				// Axis reference (process data plc/nc)
	
	// =============== About axis turque ====================
	Axis_Current_Turque 	: INT;
  	Axis_Max_Turque       	: INT;

	// ================= Sensor FeedBack ====================
  	Proximity_Switch      : DINT;
	
	// =============== Motion function blocks =================
	Axis_Power 			: MC_Power;				// FB for enable and override			[上电]
	Axis_Home			: MC_Home;				// FB for axis home						[找零]
	Axis_Reset 			: MC_Reset;				// FB to reset axis						[复位]
	Axis_Jog			: MC_Jog;				// FB to jog axis						[点动]
	Axis_Stop 			: MC_Stop;				// FB to stop axis						[停止]
	Axis_Halt			: MC_Halt;				// FB to halt axis						[停止]
	Axis_Move			: MC_MoveVelocity;		// FB to move axis (velocity movement)	[匀速运动]
	Axis_MoveAbsolute 	: MC_MoveAbsolute;		// FB to move axis absolutely			[绝对位置运动]
	Axis_MoveRelative	: MC_MoveRelative;		// FB to move axis relatively			[相对位置运动]
  	Axis_ActPosition  	: MC_ReadActualPosition;// FB to read the actual position of axis [读取电机轴的实际位置]
	Axis_ActVelocity	: MC_ReadActualVelocity;// FB to read the actual Velocity of axis [读取电机轴的实际速度]
	Axis_ExtSetPiontEnable	: MC_ExtSetPointGenEnable;	// FB to enable extsetpoint		[外部函数发生使能]
	Axis_ExtSetPiontDisable	: MC_ExtSetPointGenDisable;	// FB to disable extsetpoint	[外部函数结束使能]
  
  	// =============== Timer =================
  	Delay         : TON;          //[定时器]
END_VAR

PROPERTY ActPosition : LREAL
GET
Axis_ActPosition( Axis:= AxisRef, Enable:= TRUE );
ActPosition := Axis_ActPosition.Position;
END_GET
END_PROPERTY

PROPERTY ActVelocity : LREAL
GET
Axis_ActVelocity( Axis:= AxisRef, Enable:= TRUE,  ActualVelocity=> ActVelocity);
END_GET
END_PROPERTY

PROPERTY Current_Turque_Value : INT
GET
Current_Turque_Value := Axis_Current_Turque;
END_GET
SET
Axis_Current_Turque := Current_Turque_Value;
END_SET
END_PROPERTY

METHOD ExtSetPoint
VAR_INPUT
	Drive_ExtSetPointEnable 	: BOOL;		// 使能外部信号开始信号
	Drive_ExtSetPointDisable 	: BOOL;		// 使能外部信号结束信号
	ExSetPosition				: LREAL;	// 外部信号位置
	//Axis_Current_Turque 		: INT;		// 边界条件：丝杠位置到达两端卡死
END_VAR
// =======================外部信号发生程序==========================

IF NOT Axis_ExtSetPiontEnable.Error THEN
	Axis_ExtSetPiontEnable(	Axis:= AxisRef, 
							Execute:= Drive_ExtSetPointEnable, 
							Position:= ExSetPosition, 
							PositionType:= POSITIONTYPE_ABSOLUTE );
END_IF

IF Axis_ExtSetPiontEnable.Done THEN
	ExtSetPiontDone := 1;
	MC_ExtSetPointGenFeed(	Position:= ExSetPosition, 
							Velocity:= 10, 
							Acceleration:= 10, 
							Direction:= 1, 		// 1 = positive direction
							Axis:= AxisRef );
END_IF	

IF NOT Axis_ExtSetPiontDisable.Error THEN 
	Axis_ExtSetPiontDisable(	Axis:= AxisRef, 
								Execute:= Drive_ExtSetPointDisable);
END_IF
								
IF Axis_ExtSetPiontEnable.Error OR Axis_ExtSetPiontDisable.Error OR ABS(Axis_Current_Turque) > Axis_Max_Turque THEN
	IF Axis_ExtSetPiontEnable.Error OR Axis_ExtSetPiontDisable.Error THEN
		Axis_Error		:= TRUE;
		Axis_ErrorID 	:= Axis_Home.ErrorID;
	END_IF
	Axis_ExtSetPiontEnable(	Axis:= AxisRef, 
							Execute:= 0 );
	Axis_ExtSetPiontDisable(	Axis:= AxisRef, 
								Execute:= 1);
END_IF
END_METHOD

METHOD Halt : BOOL
VAR_INPUT
	DriveHalt		: BOOL;					// Request stop
END_VAR
// =======================电机运动停止程序==========================

IF DriveHalt THEN
	// Move Execute FALSE
	Axis_Move(	Execute	:= FALSE,
				Axis 	:= AxisRef);
ELSE
	// Reset done signal
	HaltDone := FALSE;
END_IF

// Trigger
TriggerHalt(CLK := DriveHalt);

IF TriggerHalt.Q THEN
	Axis_Halt(	Execute	:= TRUE,
				Axis 	:= AxisRef);
ELSE
	Axis_Halt(Axis := AxisRef);
END_IF

// Done / Error / Command aborted
IF Axis_Halt.Done OR Axis_Halt.Error OR Axis_Halt.CommandAborted THEN
	Axis_Error		:= Axis_Halt.Error;
	Axis_ErrorID 	:= Axis_Halt.ErrorID;
	HaltDone 		:= Axis_Halt.Done;
	
	Axis_Move(	Execute	:= FALSE,
				Axis 	:= AxisRef);
				
	Axis_Halt(	Execute	:= FALSE,
				Axis 	:= AxisRef);
END_IF

// =========================================================
END_METHOD

METHOD Home
VAR_INPUT
	//Back_Start 				: BOOL;
	//Velocity_Home	:LREAL;
	//Axis_Current_Turque 	: INT;
	Drive_Home				: BOOL;			// 找原点的信号，TURE代表还在找原点过程中
END_VAR

VAR
	//HomeSet					: BOOL;
	BackDone				: BOOL;					// 电机退回到顶点位，该标志位使能
END_VAR
// =======================找零程序==========================
// 找零程序过程为：先让丝杠回退，到达机械限位后停止,并用程序将该位置置为零位

//======================丝杠回退========================
Jog_Backward(Drive_Jog_Backward:= (Drive_Home AND (NOT BackDone)));
Jog_Velocity := Velocity_Home;
HomeDone := Axis_MoveAbsolute.Done;					// 找零结束的标志为丝杠伸长到制定距离
	
IF NOT Axis_Home.Error THEN
	IF ABS(Axis_Current_Turque) > Axis_Max_Turque AND NOT BackDone THEN
		//Drive_Home :=0;
		Jog_Backward(Drive_Jog_Backward:= 0);
		Delay(IN:= NOT Delay.Q, PT:=T#200MS, Q=> , ET=> );
		Axis_Home( 	Axis:= AxisRef, 
					Execute:= Delay.Q, 
					Position:= 0, 
					HomingMode:= MC_Direct);
		BackDone := Axis_Home.Done;				
	END_IF
	IF BackDone AND Drive_Home THEN
		Move_Absolute(Drive_Move_Absolute:= TRUE, Absolute_Position:= Home_Position );
		IF Axis_MoveAbsolute.Done THEN
			BackDone := FALSE;
			Drive_Home	:= FALSE;
		END_IF
	END_IF
END_IF

(*IF HomeSet THEN
	Jog_Backward(Drive_Jog_Backward:= 0,  Axis_Current_Turque:= Axis_Current_Turque);
	HomeDone := 1;
END_IF*)

IF Axis_Home.Error OR Axis_Home.CommandAborted OR ABS(Axis_Current_Turque) < Axis_Max_Turque THEN
	IF Axis_Jog.Error THEN
		Axis_Error		:= TRUE;
		Axis_ErrorID 	:= Axis_Home.ErrorID;
	END_IF
	Axis_Home( 	Axis:= AxisRef, 
				Execute:= FALSE);
END_IF

// =========================================================
END_METHOD

PROPERTY Home_Absolute_Position : LREAL
GET
Home_Absolute_Position := Home_Position;
END_GET
SET
Home_Position := Home_Absolute_Position;
END_SET
END_PROPERTY

METHOD Home_Sensor
VAR_INPUT
	Drive_Home				: BOOL;			// 调零使能信号
	Home_Switch				: BOOL;			// 零位调零传感器信号
	//MaxPosition_Swicth		: BOOL;
END_VAR

VAR
	//HomeSet				: BOOL;
	BackDone				: BOOL;					// 电机退回到顶点位，该标志位使能
END_VAR
// =======================找零程序==========================
// 找零程序过程为：先让丝杠回退，当传感器检测到金属表面并反馈信号后, 程序将该位置置为零位

//======================丝杠回退========================
Jog_Backward(Drive_Jog_Backward:= Drive_Home);
Jog_Velocity := Velocity_Home;
HomeDone := Axis_MoveAbsolute.Done;					// 回到零点的标志为丝杠伸长到制定距离
	
IF NOT Axis_Home.Error THEN
	IF Home_Switch AND NOT HomeDone THEN
		Drive_Home :=0;
		Jog_Backward(Drive_Jog_Backward:= Drive_Home);
		Delay(IN:= NOT Delay.Q, PT:=T#200MS, Q=> , ET=> );
		Axis_Home( 	Axis:= AxisRef, 
					Execute:= Delay.Q,
					Position:= 0, 
					HomingMode:= MC_Direct);
		BackDone := Axis_Home.Done;
	END_IF
	IF BackDone THEN
		Move_Absolute(Drive_Move_Absolute:= TRUE, Absolute_Position:= 20);
		IF Axis_MoveAbsolute.Done THEN
			BackDone := FALSE;
		END_IF
	END_IF
END_IF

(*IF HomeSet THEN
	Jog_Backward(Drive_Jog_Backward:= 0,  Axis_Current_Turque:= Axis_Current_Turque);
	HomeDone := 1;
END_IF*)

IF Axis_Home.Error OR Axis_Home.CommandAborted OR ABS(Axis_Current_Turque) < Axis_Max_Turque THEN
	IF Axis_Jog.Error THEN
		Axis_Error		:= TRUE;
		Axis_ErrorID 	:= Axis_Home.ErrorID;
	END_IF
	Axis_Home( 	Axis:= AxisRef, 
				Execute:= FALSE);
END_IF

// =========================================================
END_METHOD

METHOD Home_Sensor_Backward
VAR_INPUT
	Drive_Home				: BOOL;			// 调零使能信号
	Home_Switch				: BOOL;			// 零位调零传感器信号
	//MaxPosition_Swicth		: BOOL;
END_VAR

VAR
	//HomeSet				: BOOL;
	BackDone				: BOOL;					// 电机退回到顶点位，该标志位使能
END_VAR
// =======================找零程序==========================
// 找零程序过程为：先让丝杠回退，当传感器检测到金属表面并反馈信号后, 程序将该位置置为零位

//======================丝杠回退========================
Jog_Backward(Drive_Jog_Backward:= Drive_Home);
Jog_Velocity := Velocity_Home;
HomeDone := Axis_MoveAbsolute.Done;					// 回到零点的标志为丝杠伸长到制定距离
	
IF NOT Axis_Home.Error THEN
	IF Home_Switch THEN
		//Drive_Home :=0;
		Jog_Backward(Drive_Jog_Backward:= FALSE);
	END_IF
	
	Delay(IN:= Home_Switch AND Drive_Home, PT:=T#10MS, Q=> , ET=> );
	Axis_Home( 	Axis:= AxisRef, 
				Execute:= Delay.Q,
				Position:= 0, 
				HomingMode:= MC_Direct);
	BackDone := Axis_Home.Done;

	IF BackDone THEN
		Move_Absolute(Drive_Move_Absolute:= Drive_Home, Absolute_Position:= Home_Position);
	END_IF
	
	IF Axis_MoveAbsolute.Done THEN
			BackDone := FALSE;
	END_IF
END_IF

(*IF HomeSet THEN
	Jog_Backward(Drive_Jog_Backward:= 0,  Axis_Current_Turque:= Axis_Current_Turque);
	HomeDone := 1;
END_IF*)

IF Axis_Home.Error OR Axis_Home.CommandAborted THEN
	IF Axis_Jog.Error THEN
		Axis_Error		:= TRUE;
		Axis_ErrorID 	:= Axis_Home.ErrorID;
	END_IF
	Axis_Home( 	Axis:= AxisRef, 
				Execute:= FALSE);
END_IF

// =========================================================
END_METHOD

PROPERTY Home_Velocity : LREAL
GET
Home_Velocity := Velocity_Home;
END_GET
SET
Velocity_Home := Home_Velocity;
END_SET
END_PROPERTY

METHOD Jog_Backward
VAR_INPUT
	Drive_Jog_Backward	: BOOL;				//点动后退使能信号
	//Velocity_Jog		: LREAL;			//点动速度
	//Axis_Current_Turque : INT;				//边界条件：丝杠位置到达两端卡死
END_VAR
// =======================点动后退==========================
// 点动后退用在找零中的位置移动

IF NOT Axis_Jog.Error THEN
	Axis_Jog( 	Axis:= AxisRef, 
				JogForward:= 0, 
				JogBackwards:= Drive_Jog_Backward, 
				Mode:= MC_JOGMODE_CONTINOUS, 
				Velocity:= Velocity_Jog);
END_IF

IF Axis_Jog.Error OR Axis_Jog.CommandAborted OR ABS(Axis_Current_Turque) > Axis_Max_Turque THEN
	IF Axis_Jog.Error THEN
		Axis_Error		:= TRUE;
		Axis_ErrorID 	:= Axis_Jog.ErrorID;
	END_IF
	
	Axis_Jog(	JogForward:= 0, 
				JogBackwards:= 0, 
				Axis := AxisRef);
END_IF

(*IF ABS(Axis_Current_Turque) <1000 AND JogDone =1 THEN
	Axis_Jog(	JogForward:= 0, 
				JogBackwards:= 0, 
				Axis := AxisRef);
	JogDone :=0;
END_IF*)
				
// =========================================================
END_METHOD

METHOD Jog_Forward : BOOL
VAR_INPUT
	Drive_Jog_Forward	: BOOL;				//点动前进使能信号
	//Velocity_Jog		: LREAL;			//点动速度
	//Axis_Current_Turque : INT;				//边界条件：丝杠位置到达两端卡死
END_VAR
// =======================点动前进==========================


IF NOT Axis_Jog.Error THEN
	Axis_Jog( 	Axis:= AxisRef, 
				JogForward:= Drive_Jog_Forward, 
				JogBackwards:= 0, 
				Mode:= MC_JOGMODE_CONTINOUS, 
				Velocity:= Velocity_Jog);
END_IF

IF Axis_Jog.Error OR Axis_Jog.CommandAborted OR ABS(Axis_Current_Turque) > Axis_Max_Turque THEN
	IF Axis_Jog.Error THEN
		Axis_Error		:= TRUE;
		Axis_ErrorID 	:= Axis_Jog.ErrorID;
	END_IF
	
	Axis_Jog(	JogForward:= 0, 
				JogBackwards:= 0, 
				Axis := AxisRef);
END_IF

(*IF ABS(Axis_Current_Turque) <1000 AND JogDone =1 THEN
	Axis_Jog(	JogForward:= 0, 
				JogBackwards:= 0, 
				Axis := AxisRef);
	JogDone :=0;
END_IF*)
				
// =========================================================
END_METHOD

// =======================读写点动程序中的速度值==========================

PROPERTY Jog_Velocity : LREAL
GET
Jog_Velocity := Velocity_Jog;
END_GET
SET
Velocity_Jog := Jog_Velocity;
END_SET
END_PROPERTY

PROPERTY Max_Turque_Value : INT
SET
Axis_Max_Turque := Max_Turque_Value;
END_SET
END_PROPERTY

METHOD Move_Absolute
VAR_INPUT
	Drive_Move_Absolute : BOOL;				// 运动使能信号
	Absolute_Position	: LREAL;			// 绝对运动位置
	//Move_Velocity		: LREAL;			// 运动速度
	//Axis_Current_Turque : INT;			// 边界条件：丝杠位置到达两端卡死
END_VAR
// =======================绝对运动==========================

IF NOT Axis_MoveAbsolute.Error THEN
	Axis_MoveAbsolute(	Axis:= AxisRef, 
						Execute:= Drive_Move_Absolute, 
						Position:= Absolute_Position, 
						Velocity:= Velocity_Absolute, 
						BufferMode:= MC_Aborting );
	MoveAbsoluteDone := Axis_MoveAbsolute.Done;			// 运动到指定位置后置位
END_IF

IF Axis_MoveAbsolute.Error OR Axis_MoveAbsolute.CommandAborted OR ABS(Axis_Current_Turque) > Axis_Max_Turque THEN
	IF Axis_MoveAbsolute.Error THEN
		Axis_Error		:= TRUE;
		Axis_ErrorID 	:= Axis_MoveAbsolute.ErrorID;
	END_IF
	
	Axis_MoveAbsolute(	Axis:= AxisRef, 
						Execute:= 0, 
						BufferMode:= MC_Aborting);
END_IF

// =========================================================
END_METHOD

// =======================读写绝对运动程序中的速度值==========================

PROPERTY Move_Absolute_Velocity : LREAL
GET
Move_Absolute_Velocity := Velocity_Absolute;
END_GET
SET
Velocity_Absolute := Move_Absolute_Velocity;
END_SET
END_PROPERTY

METHOD Move_Backward
VAR_INPUT
	Move_Backward_Start : BOOL;					//匀速后退使能信号
	//Axis_Current_Turque : INT;					//边界条件：丝杠位置到达两端卡死
END_VAR
// =======================匀速后退==========================

// Not error
IF NOT Axis_Move.Error THEN
	Axis_Move(	Execute 	:= Move_Backward_Start,
				Velocity 	:= Velocity_Move,
				Direction 	:= MC_Negative_Direction,
				Axis 		:= AxisRef );
END_IF

// Error / Command aborted
IF Axis_Move.Error OR Axis_Move.CommandAborted OR ABS(Axis_Current_Turque) > Axis_Max_Turque THEN
	IF Axis_Move.Error THEN
		Axis_Error		:= TRUE;
		Axis_ErrorID 	:= Axis_Move.ErrorID;
	END_IF
	
	Axis_Move(	Execute	:= FALSE,
				Axis 	:= AxisRef);
END_IF

// =========================================================
END_METHOD

METHOD Move_Fordward
VAR_INPUT
	Move_Forward_Start : BOOL;					//匀速前进使能信号
	//Axis_Current_Turque : INT;					//边界条件：丝杠位置到达两端卡死
END_VAR
// =======================匀速前进==========================

// Not error
IF NOT Axis_Move.Error THEN
	Axis_Move(	Execute 	:= Move_Forward_Start,
				Velocity 	:= Velocity_Move,
				Direction 	:= MC_Positive_Direction,
				Axis 		:= AxisRef );
END_IF

// Error / Command aborted
IF Axis_Move.Error OR Axis_Move.CommandAborted OR ABS(Axis_Current_Turque) > Axis_Max_Turque THEN
	IF Axis_Move.Error THEN
		Axis_Error		:= TRUE;
		Axis_ErrorID 	:= Axis_Move.ErrorID;
	END_IF
	
	Axis_Move(	Execute	:= FALSE,
				Axis 	:= AxisRef);
END_IF

// =========================================================
END_METHOD

METHOD Move_Relative
VAR_INPUT
	Drive_Move_Relative		: BOOL;				// 运动使能信号
	Relative_Position		: LREAL;			// 相对运动位置
	//Move_Velocity			: LREAL;			// 运动速度
	//Axis_Current_Turque 	: INT;				// 边界条件：丝杠位置到达两端卡死
END_VAR
// =======================相对运动==========================

IF NOT Axis_MoveRelative.Error THEN
	Axis_MoveRelative(	Axis:= AxisRef, 
						Execute:= Drive_Move_Relative, 
						Distance:= Relative_Position, 
						Velocity:= Velocity_Relative, 
						BufferMode:= MC_Aborting );
END_IF

IF Axis_MoveRelative.Error OR Axis_MoveRelative.CommandAborted OR ABS(Axis_Current_Turque) > Axis_Max_Turque THEN
	IF Axis_MoveRelative.Error THEN
		Axis_Error		:= TRUE;
		Axis_ErrorID 	:= Axis_MoveRelative.ErrorID;
	END_IF
	
	Axis_MoveRelative(	Axis:= AxisRef, 
						Execute:= 0, 
						BufferMode:= MC_Aborting);
END_IF

// =========================================================
END_METHOD

// =======================读写相对运动程序中的速度值==========================

PROPERTY Move_Relative_Velocity : LREAL
GET
Move_Relative_Velocity := Velocity_Relative;
END_GET
SET
Velocity_Relative := Move_Relative_Velocity;
END_SET
END_PROPERTY

PROPERTY Move_Velocity : LREAL
GET
Move_Velocity := Velocity_Move;
END_GET
SET
Velocity_Move :=Move_Velocity :=10;
END_SET
END_PROPERTY

METHOD Power
VAR_INPUT
	Axis_Enable : BOOL;
END_VAR
// =======================上电程序==========================

Axis_Power(	Enable 			:= Axis_Enable, 
			Enable_Positive	:= Axis_Enable, 
			Enable_Negative	:= Axis_Enable, 
			Override		:= fOverride,
			Axis			:= AxisRef,
			Status			=> Power_StatusEnable);
			
IF Axis_Power.Error THEN
	Axis_Error		:= TRUE;
	Axis_ErrorID 	:= Axis_Power.ErrorID;
END_IF

AxisRef.ReadStatus();

Axis_Moves := AxisRef.Status.Moving;

// ==========================================================
END_METHOD

METHOD Reset
VAR_INPUT
	Drive_Reset		: BOOL;					// Request reset
END_VAR
// =====================驱动重置程序==========================

IF NOT Drive_Reset THEN
	ResetDone 	:= FALSE;
END_IF

// Trigger(触发器)
TriggerReset(CLK := Drive_Reset);

IF TriggerReset.Q THEN
	HaltDone 	:= FALSE;
	
	Axis_Reset(Execute := TRUE, Axis := AxisRef);
ELSE
	Axis_Reset(Axis := AxisRef);
END_IF

// Done / Error
IF Axis_Reset.Done OR Axis_Reset.Error THEN
	Axis_Error		:= Axis_Reset.Error;
	Axis_ErrorID 	:= Axis_Reset.ErrorID;
	ResetDone 		:= Axis_Reset.Done;

	Axis_Reset(	Execute	:= FALSE, Axis 	:= AxisRef);
END_IF

// =========================================================
END_METHOD

PROPERTY State_ExtSetPiontDone : BOOL
GET
State_ExtSetPiontDone := ExtSetPiontDone;
END_GET
END_PROPERTY

// =======================回零结束信号==========================

PROPERTY State_HomeDone : BOOL
GET
State_HomeDone := HomeDone;
END_GET
END_PROPERTY

// =======================点动结束信号==========================

PROPERTY State_JogDone : BOOL
GET
State_JogDone := JogDone;
END_GET
END_PROPERTY

PROPERTY State_MoveAbsoluteDone : BOOL
GET
State_MoveAbsoluteDone := MoveAbsoluteDone;
END_GET
END_PROPERTY

PROPERTY State_MoveRelativeDone : BOOL
GET
State_MoveRelativeDone := MoveRelativeDone;
END_GET
END_PROPERTY

// =======================上电状态信号==========================

PROPERTY State_PowerStatus : BOOL
GET
State_PowerStatus := Power_StatusEnable;
END_GET
END_PROPERTY

// =======================复位结束信号==========================

PROPERTY State_ResetDone : BOOL
GET
State_ResetDone := ResetDone;
END_GET
END_PROPERTY

END_FUNCTION_BLOCK

// ---- POUs/Walking_Robot_Movement.TcPOU
PROGRAM Walking_Robot_Movement
VAR_INPUT
	
	Axis_Number 			: INT;								// 定义轴数目
	
	ExSetPoint_Execute		: BOOL;								// 外部信号发生使能
	ExtSetPointEnable		: BOOL;								// 外部信号发生开始
	ExtSetPointDisable		: BOOL;								// 外部信号发生结束
	
	T_ALL					: LREAL := 40000;					// Simulink模型运动总时长
	t_Interval				: LREAL := 0.004;					// 采样时间间隔，默认为1ms
	t						: LREAL := 0;						// 当前采样时间，以0为起点
	
	// ====== Simulink模块:平地行走 ======
	Robot_Simulink			: FB_RobotWalking_OnEvenTerrain(oid:=16#01010020);
	Model_Position			: ARRAY[1..18] OF LREAL;			// Simulink中各个腿的位置
	ExSetPoint_Position		: ARRAY[1..18] OF LREAL;			// 外部信号位置
	Mapping_Position		: Variable_Model_Mapping_Control;	// 变量映射:Simulink模型->实际电机
	Mapping_Position1		: Variable_Control_Mapping_Model;	// 变量映射:检测到的实际腿位置->机器人Simulink控制模型		
	
	// ====== Simulink模块:电流滤波 =======
	Filter_Current_Simulink : FB_Filter_Current_Hexapod_Robot(oid:=16#01010030);
	Current_Turque_Filter  	: ARRAY[1..18] OF LREAL;			// 滤波后电流
	Mapping_Current_Filter	: Variable_Control_Mapping_Model;	// 变量映射:检测到的实际电流->Simulink对应电机的电流
	
	// ====== Simulink模型:触地检测 ======
	Current_Delay_Simulink	: FB_Tough_Signal_Detection_Simple(oid:=16#01010040);
	Delay_Time_1			: LREAL := 0.6;						// 延迟的时间，默认150毫秒
	MINIMUM_Current_Change	: LREAL := 150;						// 最小电流的变化值,用于判断电流变化
	Current_Change			: ARRAY[1..18] OF LREAL;			// 电流变化
	
	Current_Turque_Leg		: ARRAY[1..18] OF LREAL;			// Mapping后的电流
	
	Touch_Signal			: ARRAY [1..6] OF BOOL := [0,0,0,0,0,0];
	Touch_Signal_1			: ARRAY [1..6] OF BOOL;
	Leg_Lengths				: ARRAY [1..18] OF LREAL;
	Leg_Touch				: ARRAY [1..3] OF LREAL;
	Leg_Detection			: ARRAY [1..3] OF LREAL;
	
	// Simulink模型输入
	Step_Test				: BOOL 	:= 1;						//
	t_traj					: LREAL	:= 480;						// 行走时间
	Mode_Move				: INT	:= 1;						// 行走模式
		// 模式1 mode_move = 1,走多项式,多项式系数如下
	params_x				: ARRAY [1..5] OF LREAL := [0,0,0,0,0];
	params_y				: ARRAY [1..5] OF LREAL := [0,0,0,0,0];
	params_z				: ARRAY [1..5] OF LREAL := [0,0,0,0,0];
	
	params_alpha			: ARRAY [1..5] OF LREAL := [0,0,0,0,0]; 	// 绕Y轴
	params_beta				: ARRAY [1..5] OF LREAL := [0,0,0,0,0];	// 绕Z轴
	params_gama				: ARRAY [1..5] OF LREAL := [0,0,0,0,0];	// 绕X轴
	
		// 模式2 mode_move = 2,走圆弧,行走半径R_circle
	R_circle				: LREAL	:= 2;
	
	// Simulink模型输出
	realState				: LREAL;
	state					: LREAL;
	Number					: LREAL;
	Act_Lout				: ARRAY [1..18] OF LREAL;
	Act_Slice				: ARRAY [1..8] OF LREAL;
	Difference_Position		: ARRAY[1..18] OF LREAL;			// 实际位置与输入位置差值
		
	// 定义但未使用的变量	
	Home_Position 			: ARRAY[1..18] OF LREAL;			// Home结束后的位移值
	Current_Fiter_Delay		: ARRAY[1..18] OF LREAL;			// 延迟后的电流输出
	Difference_Current		: ARRAY[1..18] OF LREAL;			// 电流变化差值
	Mapping_Leg				: Leg_Control_Mapping_Model;		// 变量映射:实际腿->Simulink对应的腿
END_VAR

VAR
	Leg_Number				: INT;								// 定义机器人腿数
	Init_Execute			: BOOL;								// 机器人运动Simulink模型初始化使能
	Model_state: TCOM_STATE :=TCOM_STATE.TCOM_STATE_OP;
	Model_save_par			: BOOL;
END_VAR

VAR_OUTPUT
	
END_VAR


Variable_Monitor();			// 变量监测程序

Logic_Control();			// 逻辑控制程序

Variable_Set();				// 变量设定程序

Touch_Signal_Detection();	// 触地检测程序

ExSetPoint_Action();		// 外部发生程序

ACTION ExSetPoint_Action:
// ====== 模型使能 ======
IF ExSetPoint_Execute OR Walking_Robot_Control.Home_Execute THEN
	Robot_Simulink.Execute();	// Simulink模型使能
END_IF

	// 一但上电,就激活电流滤波的Simulink
IF Walking_Robot_Control.Power_Execute THEN
	Filter_Current_Simulink.Execute();
END_IF

// ====== 模型初始化 ======
IF Init_Execute THEN
	Model_state	:=TCOM_STATE.TCOM_STATE_INIT;
	t	:=0;
ELSE
	Model_state	:=TCOM_STATE.TCOM_STATE_OP;
END_IF

IF Robot_Simulink.State<>Model_state THEN
	Robot_Simulink.State	:= Model_state;
END_IF

IF NOT Model_save_par THEN
	Model_save_par:=tc3_module.SUCCEEDED(Robot_Simulink.SaveOnlineParametersForInit());
END_IF

// ====== 外部信号发生:开始运动 ======

IF ExSetPoint_Execute THEN
	FOR Axis_Number := 1 TO 18 {BY 1} DO
		Walking_Robot_Control.Axis_Robot[Axis_Number].ExtSetPoint(	Drive_ExtSetPointEnable:= ExtSetPointEnable, 
																	Drive_ExtSetPointDisable:= ExtSetPointDisable, 
																	ExSetPosition:= ExSetPoint_Position[Axis_Number]);
	END_FOR
END_IF

// ====== 外部信号发生:采样时间累加 ======
IF ExtSetPointEnable THEN	
	t := t + t_Interval;
	ExtSetPointDisable := FALSE;
END_IF

IF t>=T_ALL OR Walking_Robot_Control.Reset_Execute THEN
	ExtSetPointEnable := FALSE;
	t:=0;
	ExtSetPointDisable := TRUE;
END_IF
END_ACTION

ACTION Logic_Control:
// ====== 外部信号发生逻辑 ======
IF ExSetPoint_Execute THEN
	// 外部信号发生使能时,找零必须结束或不能找零
	Walking_Robot_Control.Home_Execute := FALSE;
	// 外部信号发生使能时,不能进行运动(特指站立,Move_Execute是站立使能)
	Walking_Robot_Control.Move_Execute := 0;		
	// 外部信号发生使能时,模型不能使能
	Init_Execute := FALSE;
ELSIF NOT ExSetPoint_Execute THEN
	// 外部信号发生不使能时,外部信号不能执行
	ExtSetPointEnable := 0;							
	ExtSetPointDisable :=0;
END_IF
IF ExtSetPointDisable THEN
	// 外部信号发生停止时,外部信号发生开始不能使能,即两者必须互斥
	ExtSetPointEnable :=0;
END_IF

	// 模型初始化时不能使能
IF 	Robot_Simulink.State = TCOM_STATE.TCOM_STATE_INIT THEN
	ExSetPoint_Execute 	:= FALSE;
END_IF

	// 找零、运动状态时,外部发生不能使能
IF Walking_Robot_Control.Home_Execute OR Walking_Robot_Control.Move_Execute THEN
	ExSetPoint_Execute := FALSE;
END_IF
END_ACTION

ACTION Safety:

END_ACTION

ACTION Touch_Signal_Detection:
// ====== 用来进行触地信号的处理 ======
// 此处已经将电流的编号由控制中的编号转换成模型中的编号

FOR Axis_Number := 1 TO 18 {BY 1} DO
	current_Delay_Simulink.stInput.Current_Filter[Axis_Number-1]		:= Current_Turque_Leg[Axis_Number];
	Current_Delay_Simulink.stInput.Delay_Time	:= Delay_Time_1;
END_FOR

current_Delay_Simulink.stInput.Number := Number;

current_Delay_Simulink.stInput.Minimum_Limit 	:= MINIMUM_Current_Change;
current_Delay_Simulink.stInput.State 			:= LREAL_TO_INT(Walking_Robot_Movement.state);
Touch_Signal_1 									:= current_Delay_Simulink.stOutput.Touch_Signal;
Walking_Robot_Movement.Leg_Touch 				:= current_Delay_Simulink.stOutput.Leg_Touch;
Walking_Robot_Movement.Leg_Detection			:= current_Delay_Simulink.stOutput.Leg_Detection;
Current_Change									:= current_Delay_Simulink.stOutput.Current_Change;

IF ExSetPoint_Execute THEN
	Current_Delay_Simulink.Execute();
END_IF
END_ACTION

ACTION Variable_Monitor:

// ====== 检测实际运动位移和输入位移差值 ======
FOR Axis_Number := 1 TO 18 {BY 1} DO
	// Walking_Robot_Control.Axis_ActPosition[] 是当前电机的实际位置
	// Mapping_Position.Controller_Leg_Variable[] 是从Simulink模型映射而来的理论上的位置
	// 另外,到目前位置(2018.5.21),Difference_Position还没有使用到
	Difference_Position[Axis_Number] := Walking_Robot_Control.Axis_ActPostion[Axis_Number]- Mapping_Position.Controller_Leg_Variable[Axis_Number]; 
END_FOR


	// 【注】:下面这段划分到Variable_Set中更好...
// ====== 电流滤波环节 ======
FOR Axis_Number := 1 TO 18 {BY 1} DO
	// 将Walking_Robot_Control中的电实际的电机电流值作为电流滤波Simulink的输入
	Filter_Current_Simulink.stInput.Current_Motor[Axis_Number-1] := Walking_Robot_Control.Current_Turque_Value[Axis_Number];
	// Current_Turque_Filter[Axis_Numer] := Filter_Current_Simulink.stInput.Current_Motor[Axis_Number-1]
END_FOR	

	// 滤波后的电机实际电流
Current_Turque_Filter := Filter_Current_Simulink.stOutput.Current_Monitor;
	
	// 电流映射: 滤波后的电机实际电流 -> 滤波后的模型对应腿电流
Mapping_Current_Filter(Controller_Leg_Variable:= Current_Turque_Filter, Model_Leg_Variable=> Current_Turque_Leg);
END_ACTION

ACTION Variable_Set:
// ====== 外部信号发生电机位置输入值 ======
FOR Axis_Number := 1 TO 18 {BY 1} DO
	// 即映射之后每隔电机的值
	ExSetPoint_Position[Axis_Number]:= Mapping_Position.Controller_Leg_Variable[Axis_Number];
END_FOR

// ====== 位置映射 ======
	// 变量映射:Simulink模型->实际电机
Mapping_Position(Model_Leg_Variable:= Model_Position);

	// 变量映射:实际电机->Simulink模型
	// 输出的Leg_Lengths目前(2018.5.21)还未使用
Mapping_Position1(Controller_Leg_Variable:= Walking_Robot_Control.Axis_ActPostion, Model_Leg_Variable=> Leg_Lengths);

Touch_Signal := Touch_Signal_1;

FOR Leg_Number := 1 TO 6 {BY 1} DO
	Robot_Simulink.stInput.Touch_Signal[Leg_Number-1]	:= BOOL_TO_LREAL(Touch_Signal[Leg_Number]);		// 传感器采集到的触地信号
END_FOR

	// 模型输入链接
Robot_Simulink.stInput.t 			:= t;					// 采样时间t与Simulink模型中的采样时间链接								
Robot_Simulink.stInput.Step_Test	:= Step_Test;			// 测试模式
Robot_simulink.stInput.params_x 	:= params_x;
Robot_simulink.stInput.params_y 	:= params_y;
Robot_simulink.stInput.params_z 	:= params_z;
Robot_simulink.stInput.params_alpha := params_alpha;
Robot_simulink.stInput.params_beta 	:= params_beta;
Robot_simulink.stInput.params_gama 	:= params_gama;
Robot_simulink.stInput.Mode_Move 	:= Mode_Move;
Robot_simulink.stInput.t_Trajectory := t_traj;
Robot_simulink.stInput.R_Circle 	:= R_circle;

	// 模型输出
Model_Position 	:= Robot_Simulink.stOutput.Disp_P;			// Simulink中的电机输出位移输入到控制模型
realState		:= Robot_Simulink.stOutput.realState;		// 模型监测状态量
state			:= Robot_Simulink.stOutput.state;			// 模型监测状态量
Number			:= Robot_Simulink.stOutput.Number;			// 已运行周期个数
Act_Slice 		:= Robot_simulink.stOutput.Act_Slice;
Act_Lout 		:= Robot_simulink.stOutput.Act_Lout;

	// 若是用户自行指定到达的地方,则使用用户指定的数据;否则,使用默认的直线
IF Walking_Welding_Robot_Control.Walking_Welding_Robot_Moving_Execute THEN
	params_x[1] := 0;
	params_x[2] := Walking_Welding_Robot_Control.Robot_Walking_Vx;
	//Params_x[2] := 0.01;
	params_x[3] := 0;
	params_x[4] := 0;
	params_x[5] := 0;
	
	params_y[1] := 0;
	params_y[2] := 0.548901719911339;
	params_y[3] := 0;
	params_y[4] := 0;
	params_y[5] := 0;
	
	params_z[1] := 0;
	params_z[2] := Walking_Welding_Robot_Control.Robot_Walking_Vz;
	//params_z[2] := 0.03;
	params_z[3] := 0;
	params_z[4] := 0;
	params_z[5] := 0;
	
	params_alpha[1] := 0;
	params_alpha[2] := Walking_Welding_Robot_Control.Robot_Walking_Va;
	//params_alpha[2] := pi/600;
	params_alpha[3] := 0;
	params_alpha[4] := 0;
	params_alpha[5] := 0;
	
	params_beta[1] := 0;
	params_beta[2] := 0;
	params_beta[3] := 0;
	params_beta[4] := 0;
	params_beta[5] := 0;
	
	params_gama[1] := 0;
	params_gama[2] := 0;
	params_gama[3] := 0;
	params_gama[4] := 0;
	params_gama[5] := 0;
ELSE
	params_x[1] := 0;
	params_x[2] := 0.01;
	params_x[3] := 0;
	params_x[4] := 0;
	params_x[5] := 0;
	
	params_y[1] := 0;
	params_y[2] := 0.548901719911339;
	params_y[3] := 0;
	params_y[4] := 0;
	params_y[5] := 0;
	
	params_z[1] := 0;
	params_z[2] := 0.03;
	params_z[3] := 0;
	params_z[4] := 0;
	params_z[5] := 0;
		
	params_alpha[1] := 0;
	params_alpha[2] := pi/600;
	params_alpha[3] := 0;
	params_alpha[4] := 0;
	params_alpha[5] := 0;
	
	params_beta[1] := 0;
	params_beta[2] := 0;
	params_beta[3] := 0;
	params_beta[4] := 0;
	params_beta[5] := 0;
	
	params_gama[1] := 0;
	params_gama[2] := 0;
	params_gama[3] := 0;
	params_gama[4] := 0;
	params_gama[5] := 0;
END_IF
END_ACTION

END_PROGRAM

// ---- DUTs/Filter_Current/FB_Filter_Current_Hexapod_Robot.TcPOU
{attribute 'TcDependOnClassFactory' := 'Filter_Current_Hexapod_Robot'}
FUNCTION_BLOCK FB_Filter_Current_Hexapod_Robot EXTENDS FB_TcMatSimObject
VAR_INPUT
	stInput: ST_Filter_Current_Hexapod_Robot_Input;
END_VAR
VAR_OUTPUT
	stOutput: ST_Filter_Current_Hexapod_Robot_Output;
END_VAR
VAR
	stInitData: ST_Filter_Current_Hexapod_Robot_InitData;
	arrDataAreas: ARRAY[1..2] OF ST_TcMatSimObjectDataAreaInfo;
	bParametersVerified: BOOL;
END_VAR

PROPERTY CallBy_Online : TctModuleCallByType
GET
hResult := GetObjPara(16#00000000,sizeof(CallBy_Online),adr(CallBy_Online));
END_GET
SET
hResult := SetObjPara(16#00000000,sizeof(CallBy_Online),adr(CallBy_Online));
END_SET
END_PROPERTY

PROPERTY CallBy_Startup : TctModuleCallByType
GET
CallBy_Startup := stInitData.CallBy;
END_GET
SET
stInitData.CallBy := CallBy_Startup;
END_SET
END_PROPERTY

PROPERTY ContextInfoArr_0_TaskCycleTimeNs_Online : UDINT
GET
hResult := GetObjPara(16#03002080,sizeof(ContextInfoArr_0_TaskCycleTimeNs_Online),adr(ContextInfoArr_0_TaskCycleTimeNs_Online));
END_GET
SET
hResult := SetObjPara(16#03002080,sizeof(ContextInfoArr_0_TaskCycleTimeNs_Online),adr(ContextInfoArr_0_TaskCycleTimeNs_Online));
END_SET
END_PROPERTY

PROPERTY ContextInfoArr_0_TaskCycleTimeNs_Startup : UDINT
GET
ContextInfoArr_0_TaskCycleTimeNs_Startup := stInitData.ContextInfoArr_0_TaskCycleTimeNs;
END_GET
SET
stInitData.ContextInfoArr_0_TaskCycleTimeNs := ContextInfoArr_0_TaskCycleTimeNs_Startup;
END_SET
END_PROPERTY

PROPERTY ContextInfoArr_0_TaskOid_Online : OTCID
GET
hResult := GetObjPara(16#03002060,sizeof(ContextInfoArr_0_TaskOid_Online),adr(ContextInfoArr_0_TaskOid_Online));
END_GET
SET
hResult := SetObjPara(16#03002060,sizeof(ContextInfoArr_0_TaskOid_Online),adr(ContextInfoArr_0_TaskOid_Online));
END_SET
END_PROPERTY

PROPERTY ContextInfoArr_0_TaskOid_Startup : OTCID
GET
ContextInfoArr_0_TaskOid_Startup := stInitData.ContextInfoArr_0_TaskOid;
END_GET
SET
stInitData.ContextInfoArr_0_TaskOid := ContextInfoArr_0_TaskOid_Startup;
END_SET
END_PROPERTY

PROPERTY ContextInfoArr_0_TaskPort_Online : UINT
GET
hResult := GetObjPara(16#03002090,sizeof(ContextInfoArr_0_TaskPort_Online),adr(ContextInfoArr_0_TaskPort_Online));
END_GET
SET
hResult := SetObjPara(16#03002090,sizeof(ContextInfoArr_0_TaskPort_Online),adr(ContextInfoArr_0_TaskPort_Online));
END_SET
END_PROPERTY

PROPERTY ContextInfoArr_0_TaskPort_Startup : UINT
GET
ContextInfoArr_0_TaskPort_Startup := stInitData.ContextInfoArr_0_TaskPort;
END_GET
SET
stInitData.ContextInfoArr_0_TaskPort := ContextInfoArr_0_TaskPort_Startup;
END_SET
END_PROPERTY

PROPERTY ContextInfoArr_0_TaskPriority_Online : UDINT
GET
hResult := GetObjPara(16#03002070,sizeof(ContextInfoArr_0_TaskPriority_Online),adr(ContextInfoArr_0_TaskPriority_Online));
END_GET
SET
hResult := SetObjPara(16#03002070,sizeof(ContextInfoArr_0_TaskPriority_Online),adr(ContextInfoArr_0_TaskPriority_Online));
END_SET
END_PROPERTY

PROPERTY ContextInfoArr_0_TaskPriority_Startup : UDINT
GET
ContextInfoArr_0_TaskPriority_Startup := stInitData.ContextInfoArr_0_TaskPriority;
END_GET
SET
stInitData.ContextInfoArr_0_TaskPriority := ContextInfoArr_0_TaskPriority_Startup;
END_SET
END_PROPERTY

PROPERTY ContextInfoArr_0_TaskSortOrder_Online : UDINT
GET
hResult := GetObjPara(16#030020b0,sizeof(ContextInfoArr_0_TaskSortOrder_Online),adr(ContextInfoArr_0_TaskSortOrder_Online));
END_GET
SET
hResult := SetObjPara(16#030020b0,sizeof(ContextInfoArr_0_TaskSortOrder_Online),adr(ContextInfoArr_0_TaskSortOrder_Online));
END_SET
END_PROPERTY

PROPERTY ContextInfoArr_0_TaskSortOrder_Startup : UDINT
GET
ContextInfoArr_0_TaskSortOrder_Startup := stInitData.ContextInfoArr_0_TaskSortOrder;
END_GET
SET
stInitData.ContextInfoArr_0_TaskSortOrder := ContextInfoArr_0_TaskSortOrder_Startup;
END_SET
END_PROPERTY

PROPERTY CycleUpdateExecuted_Online : BOOL
GET
hResult := GetObjPara(16#00000004,sizeof(CycleUpdateExecuted_Online),adr(CycleUpdateExecuted_Online));
END_GET
SET
hResult := SetObjPara(16#00000004,sizeof(CycleUpdateExecuted_Online),adr(CycleUpdateExecuted_Online));
END_SET
END_PROPERTY

METHOD Execute : HRESULT

IF (SUCCEEDED(hResult)) THEN
  hResult := VerifyParameters();
END_IF

	// update DataArea information
SetDataAreaInfo(ADR(arrDataAreas),2);
	
	// call base method
Execute := SUPER^.Execute();
END_METHOD

